LIN {X -94.212,Y -11.587,Z -73.659,A -90.000,B 90.000,C 0.000} C_DIS
LIN {X -94.293,Y -11.592,Z -73.648,A -90.000,B 90.000,C 0.000} C_DIS
LIN {X -94.845,Y -11.615,Z -73.582,A -90.000,B 90.000,C 0.000} C_DIS
LIN {X -95.072,Y -11.619,Z -73.546,A -90.000,B 90.000,C 0.000} C_DIS
LIN {X -95.448,Y -11.620,Z -73.492,A -90.000,B 90.000,C 0.000} C_DIS
LIN {X -95.686,Y -11.622,Z -73.458,A -90.000,B 90.000,C 0.000} C_DIS
LIN {X -96.285,Y -11.645,Z -73.361,A -90.000,B 90.000,C 0.000} C_DIS
LIN {X -96.529,Y -11.657,Z -73.323,A -90.000,B 90.000,C 0.000} C_DIS
LIN {X -96.718,Y -11.655,Z -73.288,A -90.000,B 90.000,C 0.000} C_DIS
LIN {X -97.124,Y -11.644,Z -73.202,A -90.000,B 90.000,C 0.000} C_DIS
LIN {X -97.511,Y -11.644,Z -73.113,A -90.000,B 90.000,C 0.000} C_DIS
LIN {X -97.707,Y -11.652,Z -73.075,A -90.000,B 90.000,C 0.000} C_DIS
LIN {X -98.138,Y -11.663,Z -72.965,A -90.000,B 90.000,C 0.000} C_DIS
LIN {X -98.421,Y -11.660,Z -72.876,A -90.000,B 90.000,C 0.000} C_DIS
LIN {X -98.629,Y -11.654,Z -72.804,A -90.000,B 90.000,C 0.000} C_DIS
LIN {X -98.764,Y -11.646,Z -72.759,A -90.000,B 90.000,C 0.000} C_DIS
LIN {X -98.907,Y -11.642,Z -72.709,A -90.000,B 90.000,C 0.000} C_DIS
LIN {X -99.025,Y -11.642,Z -72.667,A -90.000,B 90.000,C 0.000} C_DIS
LIN {X -99.303,Y -11.649,Z -72.577,A -90.000,B 90.000,C 0.000} C_DIS
LIN {X -99.385,Y -11.652,Z -72.549,A -90.000,B 90.000,C 0.000} C_DIS
LIN {X -99.802,Y -11.664,Z -72.390,A -90.000,B 90.000,C 0.000} C_DIS
LIN {X -100.084,Y -11.662,Z -72.264,A -90.000,B 90.000,C 0.000} C_DIS
LIN {X -100.297,Y -11.652,Z -72.158,A -90.000,B 90.000,C 0.000} C_DIS
LIN {X -100.506,Y -11.637,Z -72.058,A -90.000,B 90.000,C 0.000} C_DIS
LIN {X -100.618,Y -11.632,Z -72.002,A -90.000,B 90.000,C 0.000} C_DIS
LIN {X -101.008,Y -11.626,Z -71.798,A -90.000,B 90.000,C 0.000} C_DIS
LIN {X -101.217,Y -11.633,Z -71.690,A -90.000,B 90.000,C 0.000} C_DIS
LIN {X -101.505,Y -11.645,Z -71.539,A -90.000,B 90.000,C 0.000} C_DIS
LIN {X -101.784,Y -11.648,Z -71.377,A -90.000,B 90.000,C 0.000} C_DIS
LIN {X -102.159,Y -11.635,Z -71.132,A -90.000,B 90.000,C 0.000} C_DIS
LIN {X -102.376,Y -11.622,Z -70.990,A -90.000,B 90.000,C 0.000} C_DIS
LIN {X -102.782,Y -11.607,Z -70.696,A -90.000,B 90.000,C 0.000} C_DIS
LIN {X -102.971,Y -11.606,Z -70.555,A -90.000,B 90.000,C 0.000} C_DIS
LIN {X -103.503,Y -11.618,Z -70.146,A -90.000,B 90.000,C 0.000} C_DIS
LIN {X -103.891,Y -11.613,Z -69.818,A -90.000,B 90.000,C 0.000} C_DIS
LIN {X -104.471,Y -11.591,Z -69.295,A -90.000,B 90.000,C 0.000} C_DIS
LIN {X -104.553,Y -11.591,Z -69.219,A -90.000,B 90.000,C 0.000} C_DIS
LIN {X -104.963,Y -11.602,Z -68.827,A -90.000,B 90.000,C 0.000} C_DIS
LIN {X -105.136,Y -11.603,Z -68.655,A -90.000,B 90.000,C 0.000} C_DIS
LIN {X -105.249,Y -11.602,Z -68.539,A -90.000,B 90.000,C 0.000} C_DIS
LIN {X -105.573,Y -11.597,Z -68.197,A -90.000,B 90.000,C 0.000} C_DIS
LIN {X -105.950,Y -11.592,Z -67.792,A -90.000,B 90.000,C 0.000} C_DIS
LIN {X -106.246,Y -11.591,Z -67.471,A -90.000,B 90.000,C 0.000} C_DIS
LIN {X -106.503,Y -11.591,Z -67.178,A -90.000,B 90.000,C 0.000} C_DIS
LIN {X -106.747,Y -11.594,Z -66.899,A -90.000,B 90.000,C 0.000} C_DIS
LIN {X -107.149,Y -11.591,Z -66.405,A -90.000,B 90.000,C 0.000} C_DIS
LIN {X -107.576,Y -11.586,Z -65.870,A -90.000,B 90.000,C 0.000} C_DIS
LIN {X -107.870,Y -11.590,Z -65.494,A -90.000,B 90.000,C 0.000} C_DIS
LIN {X -108.183,Y -11.592,Z -65.074,A -90.000,B 90.000,C 0.000} C_DIS
LIN {X -108.727,Y -11.597,Z -64.294,A -90.000,B 90.000,C 0.000} C_DIS
LIN {X -108.884,Y -11.600,Z -64.066,A -90.000,B 90.000,C 0.000} C_DIS
LIN {X -109.086,Y -11.609,Z -63.770,A -90.000,B 90.000,C 0.000} C_DIS
LIN {X -109.795,Y -11.609,Z -62.636,A -90.000,B 90.000,C 0.000} C_DIS
LIN {X -109.878,Y -11.610,Z -62.503,A -90.000,B 90.000,C 0.000} C_DIS
LIN {X -109.980,Y -11.610,Z -62.332,A -90.000,B 90.000,C 0.000} C_DIS
LIN {X -110.151,Y -11.614,Z -62.039,A -90.000,B 90.000,C 0.000} C_DIS
LIN {X -110.277,Y -11.619,Z -61.794,A -90.000,B 90.000,C 0.000} C_DIS
LIN {X -110.690,Y -11.621,Z -60.933,A -90.000,B 90.000,C 0.000} C_DIS
LIN {X -110.735,Y -11.626,Z -60.833,A -90.000,B 90.000,C 0.000} C_DIS
LIN {X -110.921,Y -11.645,Z -60.397,A -90.000,B 90.000,C 0.000} C_DIS
LIN {X -111.213,Y -11.660,Z -59.639,A -90.000,B 90.000,C 0.000} C_DIS
LIN {X -111.406,Y -11.675,Z -59.133,A -90.000,B 90.000,C 0.000} C_DIS
LIN {X -111.465,Y -11.679,Z -58.954,A -90.000,B 90.000,C 0.000} C_DIS
LIN {X -111.561,Y -11.684,Z -58.654,A -90.000,B 90.000,C 0.000} C_DIS
LIN {X -111.600,Y -11.686,Z -58.518,A -90.000,B 90.000,C 0.000} C_DIS
LIN {X -111.705,Y -11.680,Z -58.092,A -90.000,B 90.000,C 0.000} C_DIS
LIN {X -111.798,Y -11.682,Z -57.690,A -90.000,B 90.000,C 0.000} C_DIS
LIN {X -111.872,Y -11.683,Z -57.324,A -90.000,B 90.000,C 0.000} C_DIS
LIN {X -111.987,Y -11.695,Z -56.667,A -90.000,B 90.000,C 0.000} C_DIS
LIN {X -112.103,Y -11.699,Z -56.102,A -90.000,B 90.000,C 0.000} C_DIS
LIN {X -112.133,Y -11.705,Z -55.941,A -90.000,B 90.000,C 0.000} C_DIS
LIN {X -112.214,Y -11.706,Z -55.543,A -90.000,B 90.000,C 0.000} C_DIS
LIN {X -112.258,Y -11.710,Z -55.310,A -90.000,B 90.000,C 0.000} C_DIS
LIN {X -112.301,Y -11.709,Z -55.111,A -90.000,B 90.000,C 0.000} C_DIS
LIN {X -112.331,Y -11.710,Z -54.963,A -90.000,B 90.000,C 0.000} C_DIS
LIN {X -112.384,Y -11.700,Z -54.736,A -90.000,B 90.000,C 0.000} C_DIS
LIN {X -112.413,Y -11.683,Z -54.654,A -90.000,B 90.000,C 0.000} C_DIS
LIN {X -112.468,Y -11.659,Z -54.515,A -90.000,B 90.000,C 0.000} C_DIS
LIN {X -112.573,Y -11.623,Z -54.266,A -90.000,B 90.000,C 0.000} C_DIS
LIN {X -112.724,Y -11.568,Z -53.872,A -90.000,B 90.000,C 0.000} C_DIS
LIN {X -112.828,Y -11.542,Z -53.616,A -90.000,B 90.000,C 0.000} C_DIS
LIN {X -112.987,Y -11.505,Z -53.211,A -90.000,B 90.000,C 0.000} C_DIS
LIN {X -113.167,Y -11.475,Z -52.722,A -90.000,B 90.000,C 0.000} C_DIS
LIN {X -113.273,Y -11.462,Z -52.423,A -90.000,B 90.000,C 0.000} C_DIS
LIN {X -113.396,Y -11.439,Z -52.007,A -90.000,B 90.000,C 0.000} C_DIS
LIN {X -113.436,Y -11.433,Z -51.874,A -90.000,B 90.000,C 0.000} C_DIS
LIN {X -113.514,Y -11.415,Z -51.552,A -90.000,B 90.000,C 0.000} C_DIS
LIN {X -113.736,Y -11.433,Z -51.065,A -90.000,B 90.000,C 0.000} C_DIS
LIN {X -113.844,Y -11.447,Z -50.817,A -90.000,B 90.000,C 0.000} C_DIS
LIN {X -113.954,Y -11.459,Z -50.527,A -90.000,B 90.000,C 0.000} C_DIS
LIN {X -114.109,Y -11.480,Z -50.102,A -90.000,B 90.000,C 0.000} C_DIS
LIN {X -114.142,Y -11.486,Z -50.008,A -90.000,B 90.000,C 0.000} C_DIS
LIN {X -114.248,Y -11.503,Z -49.683,A -90.000,B 90.000,C 0.000} C_DIS
LIN {X -114.317,Y -11.524,Z -49.458,A -90.000,B 90.000,C 0.000} C_DIS
LIN {X -114.400,Y -11.549,Z -49.090,A -90.000,B 90.000,C 0.000} C_DIS
LIN {X -114.487,Y -11.577,Z -48.657,A -90.000,B 90.000,C 0.000} C_DIS
LIN {X -114.535,Y -11.593,Z -48.376,A -90.000,B 90.000,C 0.000} C_DIS
LIN {X -114.551,Y -11.601,Z -48.274,A -90.000,B 90.000,C 0.000} C_DIS
LIN {X -114.562,Y -11.609,Z -48.204,A -90.000,B 90.000,C 0.000} C_DIS
LIN {X -114.587,Y -11.631,Z -47.823,A -90.000,B 90.000,C 0.000} C_DIS
LIN {X -114.597,Y -11.652,Z -47.585,A -90.000,B 90.000,C 0.000} C_DIS
LIN {X -114.602,Y -11.671,Z -47.417,A -90.000,B 90.000,C 0.000} C_DIS
LIN {X -114.599,Y -11.700,Z -47.076,A -90.000,B 90.000,C 0.000} C_DIS
LIN {X -114.573,Y -11.723,Z -46.648,A -90.000,B 90.000,C 0.000} C_DIS
LIN {X -114.555,Y -11.731,Z -46.497,A -90.000,B 90.000,C 0.000} C_DIS
LIN {X -114.524,Y -11.750,Z -46.285,A -90.000,B 90.000,C 0.000} C_DIS
LIN {X -114.446,Y -11.774,Z -45.861,A -90.000,B 90.000,C 0.000} C_DIS
LIN {X -114.403,Y -11.785,Z -45.648,A -90.000,B 90.000,C 0.000} C_DIS
LIN {X -114.366,Y -11.793,Z -45.512,A -90.000,B 90.000,C 0.000} C_DIS
LIN {X -114.304,Y -11.811,Z -45.294,A -90.000,B 90.000,C 0.000} C_DIS
LIN {X -114.182,Y -11.836,Z -44.903,A -90.000,B 90.000,C 0.000} C_DIS
LIN {X -114.168,Y -11.836,Z -44.865,A -90.000,B 90.000,C 0.000} C_DIS
LIN {X -114.169,Y -11.819,Z -44.821,A -90.000,B 90.000,C 0.000} C_DIS
LIN {X -114.168,Y -11.721,Z -44.547,A -90.000,B 90.000,C 0.000} C_DIS
LIN {X -114.165,Y -11.685,Z -44.438,A -90.000,B 90.000,C 0.000} C_DIS
LIN {X -114.151,Y -11.619,Z -44.239,A -90.000,B 90.000,C 0.000} C_DIS
LIN {X -114.122,Y -11.537,Z -43.961,A -90.000,B 90.000,C 0.000} C_DIS
LIN {X -114.106,Y -11.508,Z -43.858,A -90.000,B 90.000,C 0.000} C_DIS
LIN {X -114.085,Y -11.479,Z -43.749,A -90.000,B 90.000,C 0.000} C_DIS
LIN {X -114.038,Y -11.429,Z -43.536,A -90.000,B 90.000,C 0.000} C_DIS
LIN {X -114.035,Y -11.426,Z -43.521,A -90.000,B 90.000,C 0.000} C_DIS
LIN {X -114.241,Y -11.433,Z -43.054,A -90.000,B 90.000,C 0.000} C_DIS
LIN {X -114.306,Y -11.437,Z -42.901,A -90.000,B 90.000,C 0.000} C_DIS
LIN {X -114.518,Y -11.448,Z -42.384,A -90.000,B 90.000,C 0.000} C_DIS
LIN {X -114.643,Y -11.454,Z -42.061,A -90.000,B 90.000,C 0.000} C_DIS
LIN {X -114.710,Y -11.459,Z -41.886,A -90.000,B 90.000,C 0.000} C_DIS
LIN {X -114.857,Y -11.470,Z -41.484,A -90.000,B 90.000,C 0.000} C_DIS
LIN {X -115.017,Y -11.486,Z -40.978,A -90.000,B 90.000,C 0.000} C_DIS
LIN {X -115.171,Y -11.505,Z -40.471,A -90.000,B 90.000,C 0.000} C_DIS
LIN {X -115.237,Y -11.511,Z -40.206,A -90.000,B 90.000,C 0.000} C_DIS
LIN {X -115.269,Y -11.516,Z -40.071,A -90.000,B 90.000,C 0.000} C_DIS
LIN {X -115.346,Y -11.529,Z -39.718,A -90.000,B 90.000,C 0.000} C_DIS
LIN {X -115.399,Y -11.542,Z -39.436,A -90.000,B 90.000,C 0.000} C_DIS
LIN {X -115.423,Y -11.547,Z -39.289,A -90.000,B 90.000,C 0.000} C_DIS
LIN {X -115.469,Y -11.553,Z -38.903,A -90.000,B 90.000,C 0.000} C_DIS
LIN {X -115.487,Y -11.558,Z -38.743,A -90.000,B 90.000,C 0.000} C_DIS
LIN {X -115.510,Y -11.568,Z -38.507,A -90.000,B 90.000,C 0.000} C_DIS
LIN {X -115.536,Y -11.587,Z -38.116,A -90.000,B 90.000,C 0.000} C_DIS
LIN {X -115.547,Y -11.598,Z -37.805,A -90.000,B 90.000,C 0.000} C_DIS
LIN {X -115.546,Y -11.599,Z -37.768,A -90.000,B 90.000,C 0.000} C_DIS
LIN {X -115.535,Y -11.611,Z -37.401,A -90.000,B 90.000,C 0.000} C_DIS
LIN {X -115.517,Y -11.629,Z -37.064,A -90.000,B 90.000,C 0.000} C_DIS
LIN {X -115.474,Y -11.636,Z -36.708,A -90.000,B 90.000,C 0.000} C_DIS
LIN {X -115.454,Y -11.640,Z -36.570,A -90.000,B 90.000,C 0.000} C_DIS
LIN {X -115.407,Y -11.656,Z -36.278,A -90.000,B 90.000,C 0.000} C_DIS
LIN {X -115.349,Y -11.665,Z -35.994,A -90.000,B 90.000,C 0.000} C_DIS
LIN {X -115.297,Y -11.669,Z -35.782,A -90.000,B 90.000,C 0.000} C_DIS
LIN {X -115.179,Y -11.680,Z -35.351,A -90.000,B 90.000,C 0.000} C_DIS
LIN {X -115.107,Y -11.690,Z -35.107,A -90.000,B 90.000,C 0.000} C_DIS
LIN {X -115.003,Y -11.696,Z -34.808,A -90.000,B 90.000,C 0.000} C_DIS
LIN {X -114.904,Y -11.698,Z -34.550,A -90.000,B 90.000,C 0.000} C_DIS
LIN {X -114.796,Y -11.706,Z -34.283,A -90.000,B 90.000,C 0.000} C_DIS
LIN {X -114.748,Y -11.712,Z -34.170,A -90.000,B 90.000,C 0.000} C_DIS
LIN {X -114.623,Y -11.720,Z -33.910,A -90.000,B 90.000,C 0.000} C_DIS
LIN {X -114.429,Y -11.726,Z -33.544,A -90.000,B 90.000,C 0.000} C_DIS
LIN {X -114.375,Y -11.729,Z -33.450,A -90.000,B 90.000,C 0.000} C_DIS
LIN {X -114.266,Y -11.737,Z -33.272,A -90.000,B 90.000,C 0.000} C_DIS
LIN {X -114.093,Y -11.740,Z -33.018,A -90.000,B 90.000,C 0.000} C_DIS
LIN {X -114.019,Y -11.742,Z -32.909,A -90.000,B 90.000,C 0.000} C_DIS
LIN {X -113.928,Y -11.743,Z -32.783,A -90.000,B 90.000,C 0.000} C_DIS
LIN {X -113.839,Y -11.749,Z -32.668,A -90.000,B 90.000,C 0.000} C_DIS
LIN {X -113.552,Y -11.754,Z -32.335,A -90.000,B 90.000,C 0.000} C_DIS
LIN {X -113.377,Y -11.754,Z -32.146,A -90.000,B 90.000,C 0.000} C_DIS
LIN {X -113.255,Y -11.757,Z -32.021,A -90.000,B 90.000,C 0.000} C_DIS
LIN {X -112.860,Y -11.759,Z -31.635,A -90.000,B 90.000,C 0.000} C_DIS
LIN {X -112.787,Y -11.754,Z -31.554,A -90.000,B 90.000,C 0.000} C_DIS
LIN {X -112.743,Y -11.754,Z -31.498,A -90.000,B 90.000,C 0.000} C_DIS
LIN {X -112.607,Y -11.754,Z -31.317,A -90.000,B 90.000,C 0.000} C_DIS
LIN {X -112.172,Y -11.764,Z -30.704,A -90.000,B 90.000,C 0.000} C_DIS
LIN {X -112.046,Y -11.772,Z -30.531,A -90.000,B 90.000,C 0.000} C_DIS
LIN {X -111.786,Y -11.780,Z -30.189,A -90.000,B 90.000,C 0.000} C_DIS
LIN {X -111.636,Y -11.792,Z -29.999,A -90.000,B 90.000,C 0.000} C_DIS
LIN {X -111.260,Y -11.802,Z -29.560,A -90.000,B 90.000,C 0.000} C_DIS
LIN {X -111.118,Y -11.804,Z -29.402,A -90.000,B 90.000,C 0.000} C_DIS
LIN {X -111.007,Y -11.810,Z -29.282,A -90.000,B 90.000,C 0.000} C_DIS
LIN {X -110.702,Y -11.818,Z -28.964,A -90.000,B 90.000,C 0.000} C_DIS
LIN {X -110.630,Y -11.822,Z -28.890,A -90.000,B 90.000,C 0.000} C_DIS
LIN {X -110.226,Y -11.831,Z -28.505,A -90.000,B 90.000,C 0.000} C_DIS
LIN {X -109.683,Y -11.835,Z -28.022,A -90.000,B 90.000,C 0.000} C_DIS
LIN {X -109.483,Y -11.838,Z -27.846,A -90.000,B 90.000,C 0.000} C_DIS
LIN {X -109.036,Y -11.838,Z -27.473,A -90.000,B 90.000,C 0.000} C_DIS
LIN {X -108.440,Y -11.835,Z -27.051,A -90.000,B 90.000,C 0.000} C_DIS
LIN {X -108.173,Y -11.837,Z -26.866,A -90.000,B 90.000,C 0.000} C_DIS
LIN {X -108.077,Y -11.832,Z -26.807,A -90.000,B 90.000,C 0.000} C_DIS
LIN {X -107.401,Y -11.827,Z -26.429,A -90.000,B 90.000,C 0.000} C_DIS
LIN {X -107.170,Y -11.828,Z -26.305,A -90.000,B 90.000,C 0.000} C_DIS
LIN {X -106.974,Y -11.818,Z -26.212,A -90.000,B 90.000,C 0.000} C_DIS
LIN {X -106.880,Y -11.816,Z -26.170,A -90.000,B 90.000,C 0.000} C_DIS
LIN {X -106.375,Y -11.813,Z -25.952,A -90.000,B 90.000,C 0.000} C_DIS
LIN {X -106.083,Y -11.808,Z -25.832,A -90.000,B 90.000,C 0.000} C_DIS
LIN {X -105.983,Y -11.808,Z -25.792,A -90.000,B 90.000,C 0.000} C_DIS
LIN {X -105.685,Y -11.798,Z -25.686,A -90.000,B 90.000,C 0.000} C_DIS
LIN {X -105.383,Y -11.796,Z -25.586,A -90.000,B 90.000,C 0.000} C_DIS
LIN {X -104.972,Y -11.796,Z -25.452,A -90.000,B 90.000,C 0.000} C_DIS
LIN {X -104.611,Y -11.788,Z -25.344,A -90.000,B 90.000,C 0.000} C_DIS
LIN {X -103.526,Y -11.781,Z -25.036,A -90.000,B 90.000,C 0.000} C_DIS
LIN {X -103.108,Y -11.775,Z -24.918,A -90.000,B 90.000,C 0.000} C_DIS
LIN {X -102.960,Y -11.719,Z -24.832,A -90.000,B 90.000,C 0.000} C_DIS
LIN {X -102.802,Y -11.666,Z -24.747,A -90.000,B 90.000,C 0.000} C_DIS
LIN {X -102.662,Y -11.616,Z -24.668,A -90.000,B 90.000,C 0.000} C_DIS
LIN {X -102.539,Y -11.576,Z -24.600,A -90.000,B 90.000,C 0.000} C_DIS
LIN {X -102.363,Y -11.527,Z -24.507,A -90.000,B 90.000,C 0.000} C_DIS
LIN {X -102.114,Y -11.465,Z -24.383,A -90.000,B 90.000,C 0.000} C_DIS
LIN {X -102.014,Y -11.483,Z -24.180,A -90.000,B 90.000,C 0.000} C_DIS
LIN {X -101.901,Y -11.496,Z -23.951,A -90.000,B 90.000,C 0.000} C_DIS
LIN {X -101.819,Y -11.510,Z -23.792,A -90.000,B 90.000,C 0.000} C_DIS
LIN {X -101.710,Y -11.525,Z -23.594,A -90.000,B 90.000,C 0.000} C_DIS
LIN {X -101.650,Y -11.538,Z -23.477,A -90.000,B 90.000,C 0.000} C_DIS
LIN {X -101.419,Y -11.566,Z -23.099,A -90.000,B 90.000,C 0.000} C_DIS
LIN {X -101.286,Y -11.578,Z -22.907,A -90.000,B 90.000,C 0.000} C_DIS
LIN {X -101.230,Y -11.582,Z -22.829,A -90.000,B 90.000,C 0.000} C_DIS
LIN {X -101.083,Y -11.591,Z -22.633,A -90.000,B 90.000,C 0.000} C_DIS
LIN {X -100.905,Y -11.613,Z -22.406,A -90.000,B 90.000,C 0.000} C_DIS
LIN {X -100.650,Y -11.640,Z -22.107,A -90.000,B 90.000,C 0.000} C_DIS
LIN {X -100.625,Y -11.641,Z -22.081,A -90.000,B 90.000,C 0.000} C_DIS
LIN {X -100.490,Y -11.647,Z -21.949,A -90.000,B 90.000,C 0.000} C_DIS
LIN {X -100.295,Y -11.662,Z -21.766,A -90.000,B 90.000,C 0.000} C_DIS
LIN {X -100.058,Y -11.673,Z -21.577,A -90.000,B 90.000,C 0.000} C_DIS
LIN {X -99.895,Y -11.680,Z -21.451,A -90.000,B 90.000,C 0.000} C_DIS
LIN {X -99.709,Y -11.695,Z -21.311,A -90.000,B 90.000,C 0.000} C_DIS
LIN {X -99.552,Y -11.703,Z -21.207,A -90.000,B 90.000,C 0.000} C_DIS
LIN {X -99.332,Y -11.712,Z -21.073,A -90.000,B 90.000,C 0.000} C_DIS
LIN {X -99.161,Y -11.716,Z -20.976,A -90.000,B 90.000,C 0.000} C_DIS
LIN {X -99.058,Y -11.719,Z -20.926,A -90.000,B 90.000,C 0.000} C_DIS
LIN {X -98.927,Y -11.725,Z -20.865,A -90.000,B 90.000,C 0.000} C_DIS
LIN {X -98.675,Y -11.730,Z -20.758,A -90.000,B 90.000,C 0.000} C_DIS
LIN {X -98.528,Y -11.739,Z -20.699,A -90.000,B 90.000,C 0.000} C_DIS
LIN {X -98.215,Y -11.762,Z -20.586,A -90.000,B 90.000,C 0.000} C_DIS
LIN {X -97.800,Y -11.772,Z -20.465,A -90.000,B 90.000,C 0.000} C_DIS
LIN {X -97.726,Y -11.774,Z -20.449,A -90.000,B 90.000,C 0.000} C_DIS
LIN {X -97.685,Y -11.782,Z -20.434,A -90.000,B 90.000,C 0.000} C_DIS
LIN {X -97.660,Y -11.787,Z -20.423,A -90.000,B 90.000,C 0.000} C_DIS
LIN {X -97.342,Y -11.881,Z -20.275,A -90.000,B 90.000,C 0.000} C_DIS
LIN {X -97.307,Y -11.894,Z -20.257,A -90.000,B 90.000,C 0.000} C_DIS
LIN {X -97.142,Y -11.960,Z -20.180,A -90.000,B 90.000,C 0.000} C_DIS
LIN {X -97.021,Y -12.013,Z -20.130,A -90.000,B 90.000,C 0.000} C_DIS
LIN {X -96.913,Y -11.978,Z -19.972,A -90.000,B 90.000,C 0.000} C_DIS
LIN {X -96.868,Y -11.963,Z -19.913,A -90.000,B 90.000,C 0.000} C_DIS
LIN {X -96.756,Y -11.939,Z -19.760,A -90.000,B 90.000,C 0.000} C_DIS
LIN {X -96.712,Y -11.932,Z -19.703,A -90.000,B 90.000,C 0.000} C_DIS
LIN {X -96.487,Y -11.886,Z -19.438,A -90.000,B 90.000,C 0.000} C_DIS
LIN {X -96.353,Y -11.867,Z -19.275,A -90.000,B 90.000,C 0.000} C_DIS
LIN {X -96.154,Y -11.834,Z -19.045,A -90.000,B 90.000,C 0.000} C_DIS
LIN {X -96.089,Y -11.826,Z -18.977,A -90.000,B 90.000,C 0.000} C_DIS
LIN {X -95.848,Y -11.806,Z -18.731,A -90.000,B 90.000,C 0.000} C_DIS
LIN {X -95.599,Y -11.777,Z -18.499,A -90.000,B 90.000,C 0.000} C_DIS
LIN {X -95.498,Y -11.769,Z -18.409,A -90.000,B 90.000,C 0.000} C_DIS
LIN {X -95.397,Y -11.763,Z -18.324,A -90.000,B 90.000,C 0.000} C_DIS
LIN {X -95.266,Y -11.753,Z -18.219,A -90.000,B 90.000,C 0.000} C_DIS
LIN {X -95.101,Y -11.743,Z -18.088,A -90.000,B 90.000,C 0.000} C_DIS
LIN {X -94.938,Y -11.726,Z -17.971,A -90.000,B 90.000,C 0.000} C_DIS
LIN {X -94.819,Y -11.719,Z -17.890,A -90.000,B 90.000,C 0.000} C_DIS
LIN {X -94.307,Y -11.706,Z -17.553,A -90.000,B 90.000,C 0.000} C_DIS
LIN {X -93.957,Y -11.677,Z -17.360,A -90.000,B 90.000,C 0.000} C_DIS
LIN {X -93.803,Y -11.670,Z -17.281,A -90.000,B 90.000,C 0.000} C_DIS
LIN {X -93.404,Y -11.650,Z -17.099,A -90.000,B 90.000,C 0.000} C_DIS
LIN {X -93.140,Y -11.647,Z -16.984,A -90.000,B 90.000,C 0.000} C_DIS
LIN {X -92.940,Y -11.639,Z -16.907,A -90.000,B 90.000,C 0.000} C_DIS
LIN {X -92.233,Y -11.605,Z -16.673,A -90.000,B 90.000,C 0.000} C_DIS
LIN {X -92.077,Y -11.601,Z -16.623,A -90.000,B 90.000,C 0.000} C_DIS
LIN {X -91.780,Y -11.599,Z -16.539,A -90.000,B 90.000,C 0.000} C_DIS
LIN {X -91.315,Y -11.579,Z -16.439,A -90.000,B 90.000,C 0.000} C_DIS
LIN {X -90.900,Y -11.559,Z -16.359,A -90.000,B 90.000,C 0.000} C_DIS
LIN {X -90.731,Y -11.553,Z -16.329,A -90.000,B 90.000,C 0.000} C_DIS
LIN {X -90.367,Y -11.549,Z -16.267,A -90.000,B 90.000,C 0.000} C_DIS
LIN {X -90.191,Y -11.544,Z -16.249,A -90.000,B 90.000,C 0.000} C_DIS
LIN {X -89.833,Y -11.536,Z -16.216,A -90.000,B 90.000,C 0.000} C_DIS
LIN {X -89.165,Y -11.518,Z -16.171,A -90.000,B 90.000,C 0.000} C_DIS
LIN {X -88.792,Y -11.516,Z -16.148,A -90.000,B 90.000,C 0.000} C_DIS
LIN {X -88.664,Y -11.513,Z -16.145,A -90.000,B 90.000,C 0.000} C_DIS
LIN {X -87.183,Y -11.506,Z -16.212,A -90.000,B 90.000,C 0.000} C_DIS
LIN {X -87.099,Y -11.505,Z -16.218,A -90.000,B 90.000,C 0.000} C_DIS
LIN {X -86.917,Y -11.502,Z -16.245,A -90.000,B 90.000,C 0.000} C_DIS
LIN {X -86.828,Y -11.544,Z -16.175,A -90.000,B 90.000,C 0.000} C_DIS
LIN {X -86.636,Y -11.536,Z -15.957,A -90.000,B 90.000,C 0.000} C_DIS
LIN {X -86.604,Y -11.535,Z -15.920,A -90.000,B 90.000,C 0.000} C_DIS
LIN {X -86.521,Y -11.528,Z -15.838,A -90.000,B 90.000,C 0.000} C_DIS
LIN {X -86.433,Y -11.522,Z -15.756,A -90.000,B 90.000,C 0.000} C_DIS
LIN {X -86.245,Y -11.516,Z -15.585,A -90.000,B 90.000,C 0.000} C_DIS
LIN {X -86.143,Y -11.511,Z -15.498,A -90.000,B 90.000,C 0.000} C_DIS
LIN {X -86.001,Y -11.505,Z -15.384,A -90.000,B 90.000,C 0.000} C_DIS
LIN {X -85.716,Y -11.501,Z -15.165,A -90.000,B 90.000,C 0.000} C_DIS
LIN {X -85.489,Y -11.497,Z -15.001,A -90.000,B 90.000,C 0.000} C_DIS
LIN {X -85.292,Y -11.490,Z -14.870,A -90.000,B 90.000,C 0.000} C_DIS
LIN {X -85.056,Y -11.485,Z -14.730,A -90.000,B 90.000,C 0.000} C_DIS
LIN {X -84.838,Y -11.476,Z -14.614,A -90.000,B 90.000,C 0.000} C_DIS
LIN {X -84.643,Y -11.474,Z -14.512,A -90.000,B 90.000,C 0.000} C_DIS
LIN {X -84.496,Y -11.471,Z -14.444,A -90.000,B 90.000,C 0.000} C_DIS
LIN {X -84.276,Y -11.471,Z -14.336,A -90.000,B 90.000,C 0.000} C_DIS
LIN {X -83.945,Y -11.460,Z -14.203,A -90.000,B 90.000,C 0.000} C_DIS
LIN {X -83.789,Y -11.458,Z -14.143,A -90.000,B 90.000,C 0.000} C_DIS
LIN {X -83.679,Y -11.457,Z -14.101,A -90.000,B 90.000,C 0.000} C_DIS
LIN {X -83.236,Y -11.440,Z -13.976,A -90.000,B 90.000,C 0.000} C_DIS
LIN {X -82.907,Y -11.438,Z -13.879,A -90.000,B 90.000,C 0.000} C_DIS
LIN {X -82.511,Y -11.435,Z -13.771,A -90.000,B 90.000,C 0.000} C_DIS
LIN {X -82.198,Y -11.423,Z -13.716,A -90.000,B 90.000,C 0.000} C_DIS
LIN {X -81.975,Y -11.420,Z -13.678,A -90.000,B 90.000,C 0.000} C_DIS
LIN {X -81.855,Y -11.418,Z -13.660,A -90.000,B 90.000,C 0.000} C_DIS
LIN {X -81.523,Y -11.419,Z -13.594,A -90.000,B 90.000,C 0.000} C_DIS
LIN {X -81.089,Y -11.414,Z -13.523,A -90.000,B 90.000,C 0.000} C_DIS
LIN {X -81.051,Y -11.414,Z -13.517,A -90.000,B 90.000,C 0.000} C_DIS
LIN {X -80.708,Y -11.410,Z -13.483,A -90.000,B 90.000,C 0.000} C_DIS
LIN {X -80.352,Y -11.408,Z -13.451,A -90.000,B 90.000,C 0.000} C_DIS
LIN {X -80.279,Y -11.409,Z -13.442,A -90.000,B 90.000,C 0.000} C_DIS
LIN {X -79.938,Y -11.409,Z -13.401,A -90.000,B 90.000,C 0.000} C_DIS
LIN {X -79.461,Y -11.404,Z -13.374,A -90.000,B 90.000,C 0.000} C_DIS
LIN {X -78.870,Y -11.401,Z -13.362,A -90.000,B 90.000,C 0.000} C_DIS
LIN {X -78.618,Y -11.401,Z -13.361,A -90.000,B 90.000,C 0.000} C_DIS
LIN {X -78.465,Y -11.401,Z -13.358,A -90.000,B 90.000,C 0.000} C_DIS
LIN {X -78.196,Y -11.400,Z -13.367,A -90.000,B 90.000,C 0.000} C_DIS
LIN {X -77.753,Y -11.395,Z -13.389,A -90.000,B 90.000,C 0.000} C_DIS
LIN {X -77.193,Y -11.394,Z -13.435,A -90.000,B 90.000,C 0.000} C_DIS
LIN {X -76.796,Y -11.393,Z -13.491,A -90.000,B 90.000,C 0.000} C_DIS
LIN {X -76.319,Y -11.389,Z -13.573,A -90.000,B 90.000,C 0.000} C_DIS
LIN {X -75.821,Y -11.382,Z -13.682,A -90.000,B 90.000,C 0.000} C_DIS
LIN {X -75.289,Y -11.380,Z -13.800,A -90.000,B 90.000,C 0.000} C_DIS
LIN {X -74.826,Y -11.378,Z -13.931,A -90.000,B 90.000,C 0.000} C_DIS
LIN {X -74.667,Y -11.378,Z -13.978,A -90.000,B 90.000,C 0.000} C_DIS
LIN {X -74.204,Y -11.368,Z -14.158,A -90.000,B 90.000,C 0.000} C_DIS
LIN {X -73.840,Y -11.362,Z -14.305,A -90.000,B 90.000,C 0.000} C_DIS
LIN {X -73.396,Y -11.359,Z -14.469,A -90.000,B 90.000,C 0.000} C_DIS
LIN {X -72.945,Y -11.354,Z -14.648,A -90.000,B 90.000,C 0.000} C_DIS
LIN {X -72.686,Y -11.351,Z -14.763,A -90.000,B 90.000,C 0.000} C_DIS
LIN {X -72.170,Y -11.349,Z -14.974,A -90.000,B 90.000,C 0.000} C_DIS
LIN {X -71.784,Y -11.353,Z -15.134,A -90.000,B 90.000,C 0.000} C_DIS
LIN {X -71.617,Y -11.355,Z -15.206,A -90.000,B 90.000,C 0.000} C_DIS
LIN {X -70.795,Y -11.358,Z -15.576,A -90.000,B 90.000,C 0.000} C_DIS
LIN {X -69.979,Y -11.366,Z -15.948,A -90.000,B 90.000,C 0.000} C_DIS
LIN {X -69.569,Y -11.371,Z -16.140,A -90.000,B 90.000,C 0.000} C_DIS
LIN {X -68.609,Y -11.381,Z -16.596,A -90.000,B 90.000,C 0.000} C_DIS
LIN {X -68.413,Y -11.382,Z -16.694,A -90.000,B 90.000,C 0.000} C_DIS
LIN {X -67.117,Y -11.397,Z -17.317,A -90.000,B 90.000,C 0.000} C_DIS
LIN {X -66.418,Y -11.408,Z -17.647,A -90.000,B 90.000,C 0.000} C_DIS
LIN {X -65.864,Y -11.416,Z -17.911,A -90.000,B 90.000,C 0.000} C_DIS
LIN {X -65.636,Y -11.422,Z -18.020,A -90.000,B 90.000,C 0.000} C_DIS
LIN {X -65.398,Y -11.430,Z -18.128,A -90.000,B 90.000,C 0.000} C_DIS
LIN {X -64.927,Y -11.436,Z -18.340,A -90.000,B 90.000,C 0.000} C_DIS
LIN {X -64.688,Y -11.444,Z -18.450,A -90.000,B 90.000,C 0.000} C_DIS
LIN {X -64.411,Y -11.451,Z -18.586,A -90.000,B 90.000,C 0.000} C_DIS
LIN {X -64.115,Y -11.463,Z -18.716,A -90.000,B 90.000,C 0.000} C_DIS
LIN {X -63.630,Y -11.473,Z -18.925,A -90.000,B 90.000,C 0.000} C_DIS
LIN {X -63.453,Y -11.477,Z -19.008,A -90.000,B 90.000,C 0.000} C_DIS
LIN {X -63.283,Y -11.483,Z -19.087,A -90.000,B 90.000,C 0.000} C_DIS
LIN {X -63.009,Y -11.498,Z -19.204,A -90.000,B 90.000,C 0.000} C_DIS
LIN {X -62.543,Y -11.508,Z -19.398,A -90.000,B 90.000,C 0.000} C_DIS
LIN {X -61.955,Y -11.539,Z -19.648,A -90.000,B 90.000,C 0.000} C_DIS
LIN {X -61.221,Y -11.558,Z -19.948,A -90.000,B 90.000,C 0.000} C_DIS
LIN {X -60.878,Y -11.578,Z -20.092,A -90.000,B 90.000,C 0.000} C_DIS
LIN {X -60.186,Y -11.599,Z -20.377,A -90.000,B 90.000,C 0.000} C_DIS
LIN {X -60.084,Y -11.604,Z -20.417,A -90.000,B 90.000,C 0.000} C_DIS
LIN {X -59.308,Y -11.627,Z -20.717,A -90.000,B 90.000,C 0.000} C_DIS
LIN {X -59.119,Y -11.639,Z -20.780,A -90.000,B 90.000,C 0.000} C_DIS
LIN {X -58.731,Y -11.653,Z -20.903,A -90.000,B 90.000,C 0.000} C_DIS
LIN {X -58.424,Y -11.667,Z -21.003,A -90.000,B 90.000,C 0.000} C_DIS
LIN {X -58.280,Y -11.678,Z -21.044,A -90.000,B 90.000,C 0.000} C_DIS
LIN {X -58.100,Y -11.690,Z -21.098,A -90.000,B 90.000,C 0.000} C_DIS
LIN {X -57.688,Y -11.700,Z -21.210,A -90.000,B 90.000,C 0.000} C_DIS
LIN {X -57.102,Y -11.725,Z -21.376,A -90.000,B 90.000,C 0.000} C_DIS
LIN {X -56.796,Y -11.745,Z -21.453,A -90.000,B 90.000,C 0.000} C_DIS
LIN {X -55.966,Y -11.772,Z -21.643,A -90.000,B 90.000,C 0.000} C_DIS
LIN {X -55.467,Y -11.800,Z -21.744,A -90.000,B 90.000,C 0.000} C_DIS
LIN {X -55.234,Y -11.811,Z -21.793,A -90.000,B 90.000,C 0.000} C_DIS
LIN {X -54.619,Y -11.835,Z -21.917,A -90.000,B 90.000,C 0.000} C_DIS
LIN {X -54.475,Y -11.838,Z -21.943,A -90.000,B 90.000,C 0.000} C_DIS
LIN {X -53.703,Y -11.865,Z -22.073,A -90.000,B 90.000,C 0.000} C_DIS
LIN {X -53.054,Y -11.871,Z -22.198,A -90.000,B 90.000,C 0.000} C_DIS
LIN {X -52.704,Y -11.876,Z -22.258,A -90.000,B 90.000,C 0.000} C_DIS
LIN {X -52.048,Y -11.889,Z -22.377,A -90.000,B 90.000,C 0.000} C_DIS
LIN {X -51.623,Y -11.901,Z -22.452,A -90.000,B 90.000,C 0.000} C_DIS
LIN {X -51.222,Y -11.908,Z -22.517,A -90.000,B 90.000,C 0.000} C_DIS
LIN {X -50.846,Y -11.906,Z -22.585,A -90.000,B 90.000,C 0.000} C_DIS
LIN {X -50.087,Y -11.907,Z -22.723,A -90.000,B 90.000,C 0.000} C_DIS
LIN {X -48.722,Y -11.915,Z -22.964,A -90.000,B 90.000,C 0.000} C_DIS
LIN {X -48.419,Y -11.918,Z -23.018,A -90.000,B 90.000,C 0.000} C_DIS
LIN {X -48.134,Y -11.918,Z -23.073,A -90.000,B 90.000,C 0.000} C_DIS
LIN {X -47.344,Y -11.925,Z -23.220,A -90.000,B 90.000,C 0.000} C_DIS
LIN {X -46.745,Y -11.943,Z -23.320,A -90.000,B 90.000,C 0.000} C_DIS
LIN {X -45.133,Y -12.000,Z -23.610,A -90.000,B 90.000,C 0.000} C_DIS
LIN {X -43.319,Y -12.068,Z -23.946,A -90.000,B 90.000,C 0.000} C_DIS
LIN {X -42.916,Y -12.085,Z -24.025,A -90.000,B 90.000,C 0.000} C_DIS
LIN {X -41.975,Y -12.135,Z -24.203,A -90.000,B 90.000,C 0.000} C_DIS
LIN {X -41.789,Y -12.144,Z -24.238,A -90.000,B 90.000,C 0.000} C_DIS
LIN {X -41.373,Y -12.169,Z -24.313,A -90.000,B 90.000,C 0.000} C_DIS
LIN {X -40.647,Y -12.212,Z -24.457,A -90.000,B 90.000,C 0.000} C_DIS
LIN {X -39.432,Y -12.282,Z -24.696,A -90.000,B 90.000,C 0.000} C_DIS
LIN {X -38.120,Y -12.368,Z -24.972,A -90.000,B 90.000,C 0.000} C_DIS
LIN {X -37.996,Y -12.376,Z -24.996,A -90.000,B 90.000,C 0.000} C_DIS
LIN {X -36.939,Y -12.429,Z -25.219,A -90.000,B 90.000,C 0.000} C_DIS
LIN {X -36.164,Y -12.380,Z -25.254,A -90.000,B 90.000,C 0.000} C_DIS
LIN {X -35.887,Y -12.367,Z -25.267,A -90.000,B 90.000,C 0.000} C_DIS
LIN {X -35.659,Y -12.360,Z -25.283,A -90.000,B 90.000,C 0.000} C_DIS
LIN {X -35.168,Y -12.336,Z -25.304,A -90.000,B 90.000,C 0.000} C_DIS
LIN {X -34.302,Y -12.290,Z -25.338,A -90.000,B 90.000,C 0.000} C_DIS
LIN {X -33.603,Y -12.251,Z -25.368,A -90.000,B 90.000,C 0.000} C_DIS
LIN {X -33.499,Y -12.247,Z -25.375,A -90.000,B 90.000,C 0.000} C_DIS
LIN {X -33.134,Y -12.238,Z -25.407,A -90.000,B 90.000,C 0.000} C_DIS
LIN {X -32.384,Y -12.199,Z -25.484,A -90.000,B 90.000,C 0.000} C_DIS
LIN {X -31.917,Y -12.173,Z -25.530,A -90.000,B 90.000,C 0.000} C_DIS
LIN {X -31.511,Y -12.155,Z -25.575,A -90.000,B 90.000,C 0.000} C_DIS
LIN {X -31.190,Y -12.147,Z -25.617,A -90.000,B 90.000,C 0.000} C_DIS
LIN {X -29.446,Y -12.076,Z -25.869,A -90.000,B 90.000,C 0.000} C_DIS
LIN {X -28.314,Y -12.029,Z -26.037,A -90.000,B 90.000,C 0.000} C_DIS
LIN {X -27.260,Y -11.989,Z -26.193,A -90.000,B 90.000,C 0.000} C_DIS
LIN {X -25.187,Y -11.923,Z -26.530,A -90.000,B 90.000,C 0.000} C_DIS
LIN {X -24.913,Y -11.913,Z -26.573,A -90.000,B 90.000,C 0.000} C_DIS
LIN {X -24.278,Y -11.903,Z -26.684,A -90.000,B 90.000,C 0.000} C_DIS
LIN {X -21.916,Y -11.855,Z -27.111,A -90.000,B 90.000,C 0.000} C_DIS
LIN {X -19.911,Y -11.828,Z -27.523,A -90.000,B 90.000,C 0.000} C_DIS
LIN {X -18.700,Y -11.817,Z -27.777,A -90.000,B 90.000,C 0.000} C_DIS
LIN {X -17.522,Y -11.804,Z -28.030,A -90.000,B 90.000,C 0.000} C_DIS
LIN {X -15.964,Y -11.792,Z -28.372,A -90.000,B 90.000,C 0.000} C_DIS
LIN {X -15.554,Y -11.787,Z -28.460,A -90.000,B 90.000,C 0.000} C_DIS
LIN {X -14.898,Y -11.782,Z -28.599,A -90.000,B 90.000,C 0.000} C_DIS
LIN {X -14.261,Y -11.783,Z -28.736,A -90.000,B 90.000,C 0.000} C_DIS
LIN {X -13.540,Y -11.774,Z -28.887,A -90.000,B 90.000,C 0.000} C_DIS
LIN {X -12.125,Y -11.755,Z -29.188,A -90.000,B 90.000,C 0.000} C_DIS
LIN {X -10.507,Y -11.744,Z -29.516,A -90.000,B 90.000,C 0.000} C_DIS
LIN {X -9.808,Y -11.747,Z -29.665,A -90.000,B 90.000,C 0.000} C_DIS
LIN {X -9.254,Y -11.747,Z -29.785,A -90.000,B 90.000,C 0.000} C_DIS
LIN {X -8.609,Y -11.749,Z -29.914,A -90.000,B 90.000,C 0.000} C_DIS
LIN {X -6.213,Y -11.761,Z -30.398,A -90.000,B 90.000,C 0.000} C_DIS
LIN {X -4.810,Y -11.746,Z -30.671,A -90.000,B 90.000,C 0.000} C_DIS
LIN {X -3.119,Y -11.739,Z -31.008,A -90.000,B 90.000,C 0.000} C_DIS
LIN {X -2.367,Y -11.737,Z -31.147,A -90.000,B 90.000,C 0.000} C_DIS
LIN {X -1.289,Y -11.721,Z -31.337,A -90.000,B 90.000,C 0.000} C_DIS
LIN {X -0.397,Y -11.716,Z -31.483,A -90.000,B 90.000,C 0.000} C_DIS
LIN {X -0.045,Y -11.716,Z -31.543,A -90.000,B 90.000,C 0.000} C_DIS
LIN {X 1.093,Y -11.699,Z -31.735,A -90.000,B 90.000,C 0.000} C_DIS
LIN {X 1.657,Y -11.697,Z -31.821,A -90.000,B 90.000,C 0.000} C_DIS
LIN {X 2.714,Y -11.704,Z -31.992,A -90.000,B 90.000,C 0.000} C_DIS
LIN {X 3.458,Y -11.702,Z -32.126,A -90.000,B 90.000,C 0.000} C_DIS
LIN {X 4.753,Y -11.714,Z -32.339,A -90.000,B 90.000,C 0.000} C_DIS
LIN {X 5.409,Y -11.721,Z -32.449,A -90.000,B 90.000,C 0.000} C_DIS
LIN {X 5.651,Y -11.721,Z -32.497,A -90.000,B 90.000,C 0.000} C_DIS
LIN {X 7.337,Y -11.739,Z -32.812,A -90.000,B 90.000,C 0.000} C_DIS
LIN {X 7.728,Y -11.739,Z -32.882,A -90.000,B 90.000,C 0.000} C_DIS
LIN {X 7.983,Y -11.741,Z -32.930,A -90.000,B 90.000,C 0.000} C_DIS
LIN {X 8.349,Y -11.741,Z -33.012,A -90.000,B 90.000,C 0.000} C_DIS
LIN {X 9.214,Y -11.737,Z -33.212,A -90.000,B 90.000,C 0.000} C_DIS
LIN {X 10.580,Y -11.737,Z -33.533,A -90.000,B 90.000,C 0.000} C_DIS
LIN {X 11.985,Y -11.731,Z -33.882,A -90.000,B 90.000,C 0.000} C_DIS
LIN {X 12.404,Y -11.730,Z -33.986,A -90.000,B 90.000,C 0.000} C_DIS
LIN {X 12.803,Y -11.735,Z -34.079,A -90.000,B 90.000,C 0.000} C_DIS
LIN {X 13.234,Y -11.734,Z -34.180,A -90.000,B 90.000,C 0.000} C_DIS
LIN {X 14.351,Y -11.730,Z -34.443,A -90.000,B 90.000,C 0.000} C_DIS
LIN {X 14.549,Y -11.735,Z -34.482,A -90.000,B 90.000,C 0.000} C_DIS
LIN {X 15.657,Y -11.735,Z -34.681,A -90.000,B 90.000,C 0.000} C_DIS
LIN {X 15.848,Y -11.734,Z -34.715,A -90.000,B 90.000,C 0.000} C_DIS
LIN {X 16.161,Y -11.745,Z -34.754,A -90.000,B 90.000,C 0.000} C_DIS
LIN {X 16.763,Y -11.748,Z -34.794,A -90.000,B 90.000,C 0.000} C_DIS
LIN {X 17.292,Y -11.739,Z -34.822,A -90.000,B 90.000,C 0.000} C_DIS
LIN {X 17.449,Y -11.744,Z -34.820,A -90.000,B 90.000,C 0.000} C_DIS
LIN {X 17.784,Y -11.746,Z -34.813,A -90.000,B 90.000,C 0.000} C_DIS
LIN {X 18.506,Y -11.726,Z -34.781,A -90.000,B 90.000,C 0.000} C_DIS
LIN {X 18.584,Y -11.725,Z -34.778,A -90.000,B 90.000,C 0.000} C_DIS
LIN {X 20.055,Y -11.694,Z -34.660,A -90.000,B 90.000,C 0.000} C_DIS
LIN {X 20.960,Y -11.677,Z -34.593,A -90.000,B 90.000,C 0.000} C_DIS
LIN {X 21.137,Y -11.674,Z -34.580,A -90.000,B 90.000,C 0.000} C_DIS
LIN {X 21.254,Y -11.674,Z -34.574,A -90.000,B 90.000,C 0.000} C_DIS
LIN {X 22.361,Y -11.646,Z -34.550,A -90.000,B 90.000,C 0.000} C_DIS
LIN {X 22.818,Y -11.639,Z -34.545,A -90.000,B 90.000,C 0.000} C_DIS
LIN {X 23.000,Y -11.636,Z -34.547,A -90.000,B 90.000,C 0.000} C_DIS
LIN {X 23.842,Y -11.614,Z -34.572,A -90.000,B 90.000,C 0.000} C_DIS
LIN {X 24.145,Y -11.611,Z -34.583,A -90.000,B 90.000,C 0.000} C_DIS
LIN {X 24.593,Y -11.598,Z -34.616,A -90.000,B 90.000,C 0.000} C_DIS
LIN {X 25.301,Y -11.580,Z -34.676,A -90.000,B 90.000,C 0.000} C_DIS
LIN {X 25.817,Y -11.570,Z -34.722,A -90.000,B 90.000,C 0.000} C_DIS
LIN {X 26.060,Y -11.564,Z -34.749,A -90.000,B 90.000,C 0.000} C_DIS
LIN {X 26.608,Y -11.550,Z -34.812,A -90.000,B 90.000,C 0.000} C_DIS
LIN {X 27.338,Y -11.532,Z -34.909,A -90.000,B 90.000,C 0.000} C_DIS
LIN {X 27.464,Y -11.530,Z -34.926,A -90.000,B 90.000,C 0.000} C_DIS
LIN {X 27.764,Y -11.523,Z -34.973,A -90.000,B 90.000,C 0.000} C_DIS
LIN {X 28.165,Y -11.510,Z -35.039,A -90.000,B 90.000,C 0.000} C_DIS
LIN {X 29.192,Y -11.483,Z -35.199,A -90.000,B 90.000,C 0.000} C_DIS
LIN {X 29.573,Y -11.476,Z -35.260,A -90.000,B 90.000,C 0.000} C_DIS
LIN {X 30.521,Y -11.447,Z -35.432,A -90.000,B 90.000,C 0.000} C_DIS
LIN {X 30.960,Y -11.438,Z -35.507,A -90.000,B 90.000,C 0.000} C_DIS
LIN {X 31.495,Y -11.428,Z -35.599,A -90.000,B 90.000,C 0.000} C_DIS
LIN {X 32.649,Y -11.401,Z -35.825,A -90.000,B 90.000,C 0.000} C_DIS
LIN {X 34.012,Y -11.371,Z -36.112,A -90.000,B 90.000,C 0.000} C_DIS
LIN {X 34.323,Y -11.366,Z -36.178,A -90.000,B 90.000,C 0.000} C_DIS
LIN {X 35.984,Y -11.339,Z -36.579,A -90.000,B 90.000,C 0.000} C_DIS
LIN {X 37.654,Y -11.320,Z -37.028,A -90.000,B 90.000,C 0.000} C_DIS
LIN {X 38.405,Y -11.316,Z -37.240,A -90.000,B 90.000,C 0.000} C_DIS
LIN {X 38.865,Y -11.314,Z -37.377,A -90.000,B 90.000,C 0.000} C_DIS
LIN {X 38.958,Y -11.313,Z -37.408,A -90.000,B 90.000,C 0.000} C_DIS
LIN {X 41.274,Y -11.309,Z -38.102,A -90.000,B 90.000,C 0.000} C_DIS
LIN {X 41.465,Y -11.309,Z -38.161,A -90.000,B 90.000,C 0.000} C_DIS
LIN {X 41.501,Y -11.309,Z -38.173,A -90.000,B 90.000,C 0.000} C_DIS
LIN {X 42.574,Y -11.308,Z -38.529,A -90.000,B 90.000,C 0.000} C_DIS
LIN {X 42.574,Y -60.000,Z -38.529,A -90.000,B 90.000,C 0.000} C_DIS
LIN {X 59.471,Y -60.000,Z -47.736,A -90.000,B 90.000,C 0.000} C_DIS
LIN {X 59.471,Y -11.308,Z -47.736,A -90.000,B 90.000,C 0.000} C_DIS
LIN {X 60.087,Y -11.313,Z -48.081,A -90.000,B 90.000,C 0.000} C_DIS
LIN {X 60.291,Y -11.316,Z -48.199,A -90.000,B 90.000,C 0.000} C_DIS
LIN {X 61.211,Y -11.321,Z -48.724,A -90.000,B 90.000,C 0.000} C_DIS
LIN {X 61.757,Y -11.328,Z -49.001,A -90.000,B 90.000,C 0.000} C_DIS
LIN {X 62.522,Y -11.335,Z -49.396,A -90.000,B 90.000,C 0.000} C_DIS
LIN {X 63.426,Y -11.342,Z -49.858,A -90.000,B 90.000,C 0.000} C_DIS
LIN {X 64.165,Y -11.351,Z -50.222,A -90.000,B 90.000,C 0.000} C_DIS
LIN {X 64.623,Y -11.353,Z -50.451,A -90.000,B 90.000,C 0.000} C_DIS
LIN {X 65.310,Y -11.355,Z -50.799,A -90.000,B 90.000,C 0.000} C_DIS
LIN {X 66.461,Y -11.356,Z -51.391,A -90.000,B 90.000,C 0.000} C_DIS
LIN {X 67.054,Y -11.357,Z -51.704,A -90.000,B 90.000,C 0.000} C_DIS
LIN {X 68.566,Y -11.353,Z -52.539,A -90.000,B 90.000,C 0.000} C_DIS
LIN {X 69.039,Y -11.355,Z -52.799,A -90.000,B 90.000,C 0.000} C_DIS
LIN {X 69.800,Y -11.353,Z -53.244,A -90.000,B 90.000,C 0.000} C_DIS
LIN {X 70.742,Y -11.349,Z -53.798,A -90.000,B 90.000,C 0.000} C_DIS
LIN {X 70.993,Y -11.350,Z -53.946,A -90.000,B 90.000,C 0.000} C_DIS
LIN {X 71.846,Y -11.348,Z -54.477,A -90.000,B 90.000,C 0.000} C_DIS
LIN {X 73.095,Y -11.347,Z -55.249,A -90.000,B 90.000,C 0.000} C_DIS
LIN {X 75.176,Y -11.349,Z -56.605,A -90.000,B 90.000,C 0.000} C_DIS
LIN {X 75.577,Y -11.350,Z -56.873,A -90.000,B 90.000,C 0.000} C_DIS
LIN {X 76.930,Y -11.356,Z -57.810,A -90.000,B 90.000,C 0.000} C_DIS
LIN {X 77.395,Y -11.359,Z -58.140,A -90.000,B 90.000,C 0.000} C_DIS
LIN {X 78.611,Y -11.369,Z -59.053,A -90.000,B 90.000,C 0.000} C_DIS
LIN {X 78.742,Y -11.370,Z -59.154,A -90.000,B 90.000,C 0.000} C_DIS
LIN {X 78.742,Y -60.000,Z -59.154,A -90.000,B 90.000,C 0.000} C_DIS
LIN {X 86.813,Y -60.000,Z -48.200,A -90.000,B 90.000,C 0.000} C_DIS
LIN {X 86.813,Y -11.308,Z -48.200,A -90.000,B 90.000,C 0.000} C_DIS
LIN {X 87.471,Y -11.312,Z -47.534,A -90.000,B 90.000,C 0.000} C_DIS
LIN {X 87.493,Y -11.308,Z -47.512,A -90.000,B 90.000,C 0.000} C_DIS
LIN {X 87.493,Y -60.000,Z -47.512,A -90.000,B 90.000,C 0.000} C_DIS
LIN {X -120.015,Y -60.000,Z -240.907,A -90.000,B 90.000,C 0.000} C_DIS
LIN {X -120.015,Y -11.308,Z -240.907,A -90.000,B 90.000,C 0.000} C_DIS
LIN {X -117.247,Y -11.308,Z -239.026,A -90.000,B 90.000,C 0.000} C_DIS
LIN {X -113.998,Y -11.308,Z -236.843,A -90.000,B 90.000,C 0.000} C_DIS
LIN {X -109.848,Y -11.308,Z -234.062,A -90.000,B 90.000,C 0.000} C_DIS
LIN {X -102.156,Y -11.308,Z -228.976,A -90.000,B 90.000,C 0.000} C_DIS
LIN {X -94.210,Y -11.308,Z -223.811,A -90.000,B 90.000,C 0.000} C_DIS
LIN {X -89.135,Y -11.308,Z -220.577,A -90.000,B 90.000,C 0.000} C_DIS
LIN {X -85.949,Y -11.308,Z -218.553,A -90.000,B 90.000,C 0.000} C_DIS
LIN {X -80.440,Y -11.308,Z -215.129,A -90.000,B 90.000,C 0.000} C_DIS
LIN {X -77.455,Y -11.308,Z -213.297,A -90.000,B 90.000,C 0.000} C_DIS
LIN {X -72.390,Y -11.308,Z -210.226,A -90.000,B 90.000,C 0.000} C_DIS
LIN {X -69.847,Y -11.308,Z -208.690,A -90.000,B 90.000,C 0.000} C_DIS
LIN {X -69.311,Y -11.308,Z -208.368,A -90.000,B 90.000,C 0.000} C_DIS
LIN {X -63.361,Y -11.308,Z -204.780,A -90.000,B 90.000,C 0.000} C_DIS
LIN {X -61.539,Y -11.308,Z -203.695,A -90.000,B 90.000,C 0.000} C_DIS
LIN {X -57.313,Y -11.308,Z -201.114,A -90.000,B 90.000,C 0.000} C_DIS
LIN {X -54.615,Y -11.308,Z -199.489,A -90.000,B 90.000,C 0.000} C_DIS
LIN {X -51.668,Y -11.308,Z -197.646,A -90.000,B 90.000,C 0.000} C_DIS
LIN {X -48.905,Y -11.308,Z -195.899,A -90.000,B 90.000,C 0.000} C_DIS
LIN {X -45.943,Y -11.308,Z -193.965,A -90.000,B 90.000,C 0.000} C_DIS
LIN {X -44.127,Y -11.308,Z -192.765,A -90.000,B 90.000,C 0.000} C_DIS
LIN {X -42.146,Y -11.308,Z -191.410,A -90.000,B 90.000,C 0.000} C_DIS
LIN {X -40.431,Y -11.308,Z -190.223,A -90.000,B 90.000,C 0.000} C_DIS
LIN {X -38.656,Y -11.308,Z -188.957,A -90.000,B 90.000,C 0.000} C_DIS
LIN {X -36.959,Y -11.308,Z -187.730,A -90.000,B 90.000,C 0.000} C_DIS
LIN {X -35.437,Y -11.308,Z -186.596,A -90.000,B 90.000,C 0.000} C_DIS
LIN {X -33.756,Y -11.308,Z -185.358,A -90.000,B 90.000,C 0.000} C_DIS
LIN {X -32.322,Y -11.308,Z -184.241,A -90.000,B 90.000,C 0.000} C_DIS
LIN {X -30.852,Y -11.308,Z -183.112,A -90.000,B 90.000,C 0.000} C_DIS
LIN {X -29.435,Y -11.308,Z -181.946,A -90.000,B 90.000,C 0.000} C_DIS
LIN {X -28.470,Y -11.308,Z -181.159,A -90.000,B 90.000,C 0.000} C_DIS
LIN {X -27.157,Y -11.308,Z -179.996,A -90.000,B 90.000,C 0.000} C_DIS
LIN {X -26.033,Y -11.308,Z -179.009,A -90.000,B 90.000,C 0.000} C_DIS
LIN {X -24.010,Y -11.308,Z -177.055,A -90.000,B 90.000,C 0.000} C_DIS
LIN {X -23.302,Y -11.308,Z -176.288,A -90.000,B 90.000,C 0.000} C_DIS
LIN {X -22.118,Y -11.308,Z -175.018,A -90.000,B 90.000,C 0.000} C_DIS
LIN {X -21.400,Y -11.308,Z -174.130,A -90.000,B 90.000,C 0.000} C_DIS
LIN {X -20.526,Y -11.308,Z -173.070,A -90.000,B 90.000,C 0.000} C_DIS
LIN {X -19.980,Y -11.308,Z -172.290,A -90.000,B 90.000,C 0.000} C_DIS
LIN {X -19.037,Y -11.308,Z -170.976,A -90.000,B 90.000,C 0.000} C_DIS
LIN {X -18.248,Y -11.308,Z -169.695,A -90.000,B 90.000,C 0.000} C_DIS
LIN {X -17.681,Y -11.308,Z -168.755,A -90.000,B 90.000,C 0.000} C_DIS
LIN {X -16.910,Y -11.308,Z -167.280,A -90.000,B 90.000,C 0.000} C_DIS
LIN {X -16.482,Y -11.308,Z -166.456,A -90.000,B 90.000,C 0.000} C_DIS
LIN {X -15.851,Y -11.308,Z -164.959,A -90.000,B 90.000,C 0.000} C_DIS
LIN {X -15.638,Y -11.308,Z -164.459,A -90.000,B 90.000,C 0.000} C_DIS
LIN {X -15.239,Y -11.308,Z -163.088,A -90.000,B 90.000,C 0.000} C_DIS
LIN {X -15.179,Y -11.308,Z -162.892,A -90.000,B 90.000,C 0.000} C_DIS
LIN {X -15.106,Y -11.308,Z -162.060,A -90.000,B 90.000,C 0.000} C_DIS
LIN {X -15.162,Y -11.308,Z -161.680,A -90.000,B 90.000,C 0.000} C_DIS
LIN {X -15.177,Y -11.308,Z -161.560,A -90.000,B 90.000,C 0.000} C_DIS
LIN {X -15.242,Y -11.308,Z -161.392,A -90.000,B 90.000,C 0.000} C_DIS
LIN {X -15.380,Y -11.308,Z -160.998,A -90.000,B 90.000,C 0.000} C_DIS
LIN {X -15.558,Y -11.308,Z -160.681,A -90.000,B 90.000,C 0.000} C_DIS
LIN {X -15.594,Y -11.308,Z -160.606,A -90.000,B 90.000,C 0.000} C_DIS
LIN {X -15.823,Y -11.308,Z -160.137,A -90.000,B 90.000,C 0.000} C_DIS
LIN {X -16.234,Y -11.308,Z -159.462,A -90.000,B 90.000,C 0.000} C_DIS
LIN {X -16.407,Y -11.308,Z -159.131,A -90.000,B 90.000,C 0.000} C_DIS
LIN {X -16.816,Y -11.308,Z -158.560,A -90.000,B 90.000,C 0.000} C_DIS
LIN {X -17.079,Y -11.308,Z -158.163,A -90.000,B 90.000,C 0.000} C_DIS
LIN {X -17.206,Y -11.308,Z -157.959,A -90.000,B 90.000,C 0.000} C_DIS
LIN {X -17.736,Y -11.308,Z -157.326,A -90.000,B 90.000,C 0.000} C_DIS
LIN {X -18.008,Y -11.308,Z -156.997,A -90.000,B 90.000,C 0.000} C_DIS
LIN {X -18.359,Y -11.308,Z -156.535,A -90.000,B 90.000,C 0.000} C_DIS
LIN {X -19.534,Y -11.308,Z -155.295,A -90.000,B 90.000,C 0.000} C_DIS
LIN {X -19.847,Y -11.308,Z -154.953,A -90.000,B 90.000,C 0.000} C_DIS
LIN {X -20.098,Y -11.308,Z -154.670,A -90.000,B 90.000,C 0.000} C_DIS
LIN {X -21.956,Y -11.308,Z -152.876,A -90.000,B 90.000,C 0.000} C_DIS
LIN {X -22.691,Y -11.308,Z -152.133,A -90.000,B 90.000,C 0.000} C_DIS
LIN {X -24.880,Y -11.308,Z -149.981,A -90.000,B 90.000,C 0.000} C_DIS
LIN {X -25.774,Y -11.308,Z -149.070,A -90.000,B 90.000,C 0.000} C_DIS
LIN {X -28.039,Y -11.308,Z -146.647,A -90.000,B 90.000,C 0.000} C_DIS
LIN {X -28.646,Y -11.308,Z -145.992,A -90.000,B 90.000,C 0.000} C_DIS
LIN {X -29.080,Y -11.308,Z -145.514,A -90.000,B 90.000,C 0.000} C_DIS
LIN {X -29.302,Y -11.308,Z -145.261,A -90.000,B 90.000,C 0.000} C_DIS
LIN {X -29.397,Y -11.308,Z -145.146,A -90.000,B 90.000,C 0.000} C_DIS
LIN {X -32.088,Y -11.308,Z -141.796,A -90.000,B 90.000,C 0.000} C_DIS
LIN {X -32.424,Y -11.308,Z -141.370,A -90.000,B 90.000,C 0.000} C_DIS
LIN {X -32.702,Y -11.308,Z -140.971,A -90.000,B 90.000,C 0.000} C_DIS
LIN {X -32.969,Y -11.308,Z -140.540,A -90.000,B 90.000,C 0.000} C_DIS
LIN {X -35.246,Y -11.308,Z -136.931,A -90.000,B 90.000,C 0.000} C_DIS
LIN {X -35.482,Y -11.308,Z -136.505,A -90.000,B 90.000,C 0.000} C_DIS
LIN {X -36.550,Y -11.308,Z -134.456,A -90.000,B 90.000,C 0.000} C_DIS
LIN {X -37.577,Y -11.308,Z -132.478,A -90.000,B 90.000,C 0.000} C_DIS
LIN {X -39.277,Y -11.308,Z -128.695,A -90.000,B 90.000,C 0.000} C_DIS
LIN {X -39.403,Y -11.308,Z -128.407,A -90.000,B 90.000,C 0.000} C_DIS
LIN {X -40.872,Y -11.308,Z -124.859,A -90.000,B 90.000,C 0.000} C_DIS
LIN {X -41.656,Y -11.308,Z -123.002,A -90.000,B 90.000,C 0.000} C_DIS
LIN {X -41.916,Y -11.308,Z -122.444,A -90.000,B 90.000,C 0.000} C_DIS
LIN {X -42.357,Y -11.308,Z -121.509,A -90.000,B 90.000,C 0.000} C_DIS
LIN {X -43.080,Y -11.308,Z -120.253,A -90.000,B 90.000,C 0.000} C_DIS
LIN {X -43.814,Y -11.308,Z -119.207,A -90.000,B 90.000,C 0.000} C_DIS
LIN {X -44.088,Y -11.308,Z -118.815,A -90.000,B 90.000,C 0.000} C_DIS
LIN {X -44.337,Y -11.308,Z -118.497,A -90.000,B 90.000,C 0.000} C_DIS
LIN {X -45.753,Y -11.308,Z -116.718,A -90.000,B 90.000,C 0.000} C_DIS
LIN {X -48.567,Y -11.308,Z -113.314,A -90.000,B 90.000,C 0.000} C_DIS
LIN {X -49.660,Y -11.308,Z -111.991,A -90.000,B 90.000,C 0.000} C_DIS
LIN {X -50.187,Y -11.308,Z -111.359,A -90.000,B 90.000,C 0.000} C_DIS
LIN {X -51.679,Y -11.308,Z -109.496,A -90.000,B 90.000,C 0.000} C_DIS
LIN {X -52.643,Y -11.308,Z -108.298,A -90.000,B 90.000,C 0.000} C_DIS
LIN {X -55.067,Y -11.308,Z -105.083,A -90.000,B 90.000,C 0.000} C_DIS
LIN {X -57.439,Y -11.308,Z -101.855,A -90.000,B 90.000,C 0.000} C_DIS
LIN {X -58.836,Y -11.308,Z -99.974,A -90.000,B 90.000,C 0.000} C_DIS
LIN {X -59.601,Y -11.308,Z -98.941,A -90.000,B 90.000,C 0.000} C_DIS
LIN {X -60.315,Y -11.308,Z -98.039,A -90.000,B 90.000,C 0.000} C_DIS
LIN {X -61.463,Y -11.308,Z -96.581,A -90.000,B 90.000,C 0.000} C_DIS
LIN {X -61.816,Y -11.308,Z -96.122,A -90.000,B 90.000,C 0.000} C_DIS
LIN {X -63.208,Y -11.308,Z -94.561,A -90.000,B 90.000,C 0.000} C_DIS
LIN {X -63.751,Y -11.308,Z -93.930,A -90.000,B 90.000,C 0.000} C_DIS
LIN {X -65.336,Y -11.308,Z -92.364,A -90.000,B 90.000,C 0.000} C_DIS
LIN {X -65.630,Y -11.308,Z -92.059,A -90.000,B 90.000,C 0.000} C_DIS
LIN {X -66.839,Y -11.308,Z -91.004,A -90.000,B 90.000,C 0.000} C_DIS
LIN {X -67.505,Y -11.308,Z -90.394,A -90.000,B 90.000,C 0.000} C_DIS
LIN {X -69.109,Y -11.308,Z -89.139,A -90.000,B 90.000,C 0.000} C_DIS
LIN {X -69.467,Y -11.308,Z -88.848,A -90.000,B 90.000,C 0.000} C_DIS
LIN {X -69.989,Y -11.308,Z -88.463,A -90.000,B 90.000,C 0.000} C_DIS
LIN {X -71.693,Y -11.308,Z -87.240,A -90.000,B 90.000,C 0.000} C_DIS
LIN {X -72.321,Y -11.308,Z -86.810,A -90.000,B 90.000,C 0.000} C_DIS
LIN {X -73.520,Y -11.308,Z -86.005,A -90.000,B 90.000,C 0.000} C_DIS
LIN {X -74.178,Y -11.308,Z -85.579,A -90.000,B 90.000,C 0.000} C_DIS
LIN {X -75.638,Y -11.308,Z -84.644,A -90.000,B 90.000,C 0.000} C_DIS
LIN {X -77.567,Y -11.308,Z -83.441,A -90.000,B 90.000,C 0.000} C_DIS
LIN {X -79.204,Y -11.308,Z -82.416,A -90.000,B 90.000,C 0.000} C_DIS
LIN {X -80.404,Y -11.308,Z -81.632,A -90.000,B 90.000,C 0.000} C_DIS
LIN {X -80.979,Y -11.308,Z -81.244,A -90.000,B 90.000,C 0.000} C_DIS
LIN {X -81.834,Y -11.308,Z -80.650,A -90.000,B 90.000,C 0.000} C_DIS
LIN {X -82.183,Y -11.308,Z -80.399,A -90.000,B 90.000,C 0.000} C_DIS
LIN {X -83.154,Y -11.308,Z -79.660,A -90.000,B 90.000,C 0.000} C_DIS
LIN {X -83.627,Y -11.308,Z -79.285,A -90.000,B 90.000,C 0.000} C_DIS
LIN {X -84.622,Y -11.308,Z -78.444,A -90.000,B 90.000,C 0.000} C_DIS
LIN {X -85.571,Y -11.308,Z -77.608,A -90.000,B 90.000,C 0.000} C_DIS
LIN {X -86.476,Y -11.308,Z -76.828,A -90.000,B 90.000,C 0.000} C_DIS
LIN {X -87.053,Y -11.308,Z -76.372,A -90.000,B 90.000,C 0.000} C_DIS
LIN {X -87.757,Y -11.308,Z -75.901,A -90.000,B 90.000,C 0.000} C_DIS
LIN {X -88.530,Y -11.308,Z -75.455,A -90.000,B 90.000,C 0.000} C_DIS
LIN {X -89.073,Y -11.308,Z -75.180,A -90.000,B 90.000,C 0.000} C_DIS
LIN {X -89.939,Y -11.308,Z -74.790,A -90.000,B 90.000,C 0.000} C_DIS
LIN {X -90.389,Y -11.308,Z -74.607,A -90.000,B 90.000,C 0.000} C_DIS
LIN {X -90.941,Y -11.308,Z -74.405,A -90.000,B 90.000,C 0.000} C_DIS
LIN {X -91.030,Y -11.308,Z -74.374,A -90.000,B 90.000,C 0.000} C_DIS
LIN {X -91.527,Y -11.308,Z -74.217,A -90.000,B 90.000,C 0.000} C_DIS
LIN {X -91.764,Y -11.308,Z -74.153,A -90.000,B 90.000,C 0.000} C_DIS
LIN {X -92.042,Y -11.308,Z -74.095,A -90.000,B 90.000,C 0.000} C_DIS
LIN {X -92.439,Y -11.308,Z -74.029,A -90.000,B 90.000,C 0.000} C_DIS
LIN {X -93.173,Y -11.308,Z -73.932,A -90.000,B 90.000,C 0.000} C_DIS
LIN {X -93.645,Y -11.308,Z -73.895,A -90.000,B 90.000,C 0.000} C_DIS
LIN {X -94.140,Y -11.308,Z -73.831,A -90.000,B 90.000,C 0.000} C_DIS
LIN {X -95.058,Y -11.308,Z -73.746,A -90.000,B 90.000,C 0.000} C_DIS
LIN {X -95.568,Y -11.308,Z -73.674,A -90.000,B 90.000,C 0.000} C_DIS
LIN {X -95.931,Y -11.308,Z -73.620,A -90.000,B 90.000,C 0.000} C_DIS
LIN {X -96.047,Y -11.308,Z -73.610,A -90.000,B 90.000,C 0.000} C_DIS
LIN {X -96.452,Y -11.308,Z -73.561,A -90.000,B 90.000,C 0.000} C_DIS
LIN {X -96.731,Y -11.308,Z -73.508,A -90.000,B 90.000,C 0.000} C_DIS
LIN {X -97.171,Y -11.308,Z -73.404,A -90.000,B 90.000,C 0.000} C_DIS
LIN {X -97.637,Y -11.308,Z -73.327,A -90.000,B 90.000,C 0.000} C_DIS
LIN {X -98.066,Y -11.308,Z -73.225,A -90.000,B 90.000,C 0.000} C_DIS
LIN {X -98.349,Y -11.308,Z -73.133,A -90.000,B 90.000,C 0.000} C_DIS
LIN {X -98.675,Y -11.308,Z -73.014,A -90.000,B 90.000,C 0.000} C_DIS
LIN {X -99.322,Y -11.308,Z -72.816,A -90.000,B 90.000,C 0.000} C_DIS
LIN {X -99.737,Y -11.308,Z -72.666,A -90.000,B 90.000,C 0.000} C_DIS
LIN {X -100.020,Y -11.308,Z -72.539,A -90.000,B 90.000,C 0.000} C_DIS
LIN {X -100.604,Y -11.308,Z -72.228,A -90.000,B 90.000,C 0.000} C_DIS
LIN {X -101.164,Y -11.308,Z -71.956,A -90.000,B 90.000,C 0.000} C_DIS
LIN {X -101.454,Y -11.308,Z -71.812,A -90.000,B 90.000,C 0.000} C_DIS
LIN {X -101.732,Y -11.308,Z -71.653,A -90.000,B 90.000,C 0.000} C_DIS
LIN {X -102.109,Y -11.308,Z -71.397,A -90.000,B 90.000,C 0.000} C_DIS
LIN {X -102.628,Y -11.308,Z -71.037,A -90.000,B 90.000,C 0.000} C_DIS
LIN {X -103.467,Y -11.308,Z -70.406,A -90.000,B 90.000,C 0.000} C_DIS
LIN {X -103.814,Y -11.308,Z -70.110,A -90.000,B 90.000,C 0.000} C_DIS
LIN {X -104.131,Y -11.308,Z -69.836,A -90.000,B 90.000,C 0.000} C_DIS
LIN {X -105.146,Y -11.308,Z -68.890,A -90.000,B 90.000,C 0.000} C_DIS
LIN {X -105.491,Y -11.308,Z -68.525,A -90.000,B 90.000,C 0.000} C_DIS
LIN {X -106.444,Y -11.308,Z -67.489,A -90.000,B 90.000,C 0.000} C_DIS
LIN {X -106.721,Y -11.308,Z -67.174,A -90.000,B 90.000,C 0.000} C_DIS
LIN {X -107.296,Y -11.308,Z -66.468,A -90.000,B 90.000,C 0.000} C_DIS
LIN {X -107.849,Y -11.308,Z -65.768,A -90.000,B 90.000,C 0.000} C_DIS
LIN {X -108.123,Y -11.308,Z -65.404,A -90.000,B 90.000,C 0.000} C_DIS
LIN {X -108.806,Y -11.308,Z -64.465,A -90.000,B 90.000,C 0.000} C_DIS
LIN {X -109.073,Y -11.308,Z -64.084,A -90.000,B 90.000,C 0.000} C_DIS
LIN {X -109.874,Y -11.308,Z -62.803,A -90.000,B 90.000,C 0.000} C_DIS
LIN {X -110.263,Y -11.308,Z -62.153,A -90.000,B 90.000,C 0.000} C_DIS
LIN {X -110.774,Y -11.308,Z -61.179,A -90.000,B 90.000,C 0.000} C_DIS
LIN {X -110.962,Y -11.308,Z -60.763,A -90.000,B 90.000,C 0.000} C_DIS
LIN {X -111.468,Y -11.308,Z -59.492,A -90.000,B 90.000,C 0.000} C_DIS
LIN {X -111.566,Y -11.308,Z -59.220,A -90.000,B 90.000,C 0.000} C_DIS
LIN {X -111.720,Y -11.308,Z -58.779,A -90.000,B 90.000,C 0.000} C_DIS
LIN {X -111.870,Y -11.308,Z -58.274,A -90.000,B 90.000,C 0.000} C_DIS
LIN {X -112.012,Y -11.308,Z -57.796,A -90.000,B 90.000,C 0.000} C_DIS
LIN {X -112.028,Y -11.308,Z -57.728,A -90.000,B 90.000,C 0.000} C_DIS
LIN {X -112.122,Y -11.308,Z -57.282,A -90.000,B 90.000,C 0.000} C_DIS
LIN {X -112.252,Y -11.308,Z -56.574,A -90.000,B 90.000,C 0.000} C_DIS
LIN {X -112.349,Y -11.308,Z -56.108,A -90.000,B 90.000,C 0.000} C_DIS
LIN {X -112.398,Y -11.308,Z -55.844,A -90.000,B 90.000,C 0.000} C_DIS
LIN {X -112.484,Y -11.308,Z -55.453,A -90.000,B 90.000,C 0.000} C_DIS
LIN {X -112.506,Y -11.308,Z -55.365,A -90.000,B 90.000,C 0.000} C_DIS
LIN {X -112.664,Y -11.308,Z -54.669,A -90.000,B 90.000,C 0.000} C_DIS
LIN {X -112.877,Y -11.308,Z -53.941,A -90.000,B 90.000,C 0.000} C_DIS
LIN {X -113.178,Y -11.308,Z -53.024,A -90.000,B 90.000,C 0.000} C_DIS
LIN {X -113.360,Y -11.308,Z -52.461,A -90.000,B 90.000,C 0.000} C_DIS
LIN {X -113.502,Y -11.308,Z -51.915,A -90.000,B 90.000,C 0.000} C_DIS
LIN {X -113.595,Y -11.308,Z -51.469,A -90.000,B 90.000,C 0.000} C_DIS
LIN {X -113.599,Y -11.308,Z -51.445,A -90.000,B 90.000,C 0.000} C_DIS
LIN {X -113.782,Y -11.308,Z -51.057,A -90.000,B 90.000,C 0.000} C_DIS
LIN {X -113.939,Y -11.308,Z -50.706,A -90.000,B 90.000,C 0.000} C_DIS
LIN {X -114.114,Y -11.308,Z -50.263,A -90.000,B 90.000,C 0.000} C_DIS
LIN {X -114.263,Y -11.308,Z -49.868,A -90.000,B 90.000,C 0.000} C_DIS
LIN {X -114.434,Y -11.308,Z -49.373,A -90.000,B 90.000,C 0.000} C_DIS
LIN {X -114.463,Y -11.308,Z -49.286,A -90.000,B 90.000,C 0.000} C_DIS
LIN {X -114.561,Y -11.308,Z -48.902,A -90.000,B 90.000,C 0.000} C_DIS
LIN {X -114.667,Y -11.308,Z -48.448,A -90.000,B 90.000,C 0.000} C_DIS
LIN {X -114.763,Y -11.308,Z -47.970,A -90.000,B 90.000,C 0.000} C_DIS
LIN {X -114.845,Y -11.308,Z -47.135,A -90.000,B 90.000,C 0.000} C_DIS
LIN {X -114.859,Y -11.308,Z -46.765,A -90.000,B 90.000,C 0.000} C_DIS
LIN {X -114.849,Y -11.308,Z -46.324,A -90.000,B 90.000,C 0.000} C_DIS
LIN {X -114.819,Y -11.308,Z -45.943,A -90.000,B 90.000,C 0.000} C_DIS
LIN {X -114.756,Y -11.308,Z -45.485,A -90.000,B 90.000,C 0.000} C_DIS
LIN {X -114.716,Y -11.308,Z -45.273,A -90.000,B 90.000,C 0.000} C_DIS
LIN {X -114.635,Y -11.308,Z -44.907,A -90.000,B 90.000,C 0.000} C_DIS
LIN {X -114.530,Y -11.308,Z -44.496,A -90.000,B 90.000,C 0.000} C_DIS
LIN {X -114.412,Y -11.308,Z -44.152,A -90.000,B 90.000,C 0.000} C_DIS
LIN {X -114.260,Y -11.308,Z -43.756,A -90.000,B 90.000,C 0.000} C_DIS
LIN {X -114.113,Y -11.308,Z -43.434,A -90.000,B 90.000,C 0.000} C_DIS
LIN {X -114.374,Y -11.308,Z -42.849,A -90.000,B 90.000,C 0.000} C_DIS
LIN {X -114.630,Y -11.308,Z -42.238,A -90.000,B 90.000,C 0.000} C_DIS
LIN {X -114.811,Y -11.308,Z -41.776,A -90.000,B 90.000,C 0.000} C_DIS
LIN {X -114.976,Y -11.308,Z -41.322,A -90.000,B 90.000,C 0.000} C_DIS
LIN {X -115.167,Y -11.308,Z -40.736,A -90.000,B 90.000,C 0.000} C_DIS
LIN {X -115.298,Y -11.308,Z -40.319,A -90.000,B 90.000,C 0.000} C_DIS
LIN {X -115.387,Y -11.308,Z -39.952,A -90.000,B 90.000,C 0.000} C_DIS
LIN {X -115.493,Y -11.308,Z -39.497,A -90.000,B 90.000,C 0.000} C_DIS
LIN {X -115.558,Y -11.308,Z -39.145,A -90.000,B 90.000,C 0.000} C_DIS
LIN {X -115.642,Y -11.308,Z -38.476,A -90.000,B 90.000,C 0.000} C_DIS
LIN {X -115.657,Y -11.308,Z -38.346,A -90.000,B 90.000,C 0.000} C_DIS
LIN {X -115.695,Y -11.308,Z -37.922,A -90.000,B 90.000,C 0.000} C_DIS
LIN {X -115.707,Y -11.308,Z -37.619,A -90.000,B 90.000,C 0.000} C_DIS
LIN {X -115.701,Y -11.308,Z -37.164,A -90.000,B 90.000,C 0.000} C_DIS
LIN {X -115.689,Y -11.308,Z -36.861,A -90.000,B 90.000,C 0.000} C_DIS
LIN {X -115.598,Y -11.308,Z -36.120,A -90.000,B 90.000,C 0.000} C_DIS
LIN {X -115.543,Y -11.308,Z -35.841,A -90.000,B 90.000,C 0.000} C_DIS
LIN {X -115.462,Y -11.308,Z -35.496,A -90.000,B 90.000,C 0.000} C_DIS
LIN {X -115.365,Y -11.308,Z -35.122,A -90.000,B 90.000,C 0.000} C_DIS
LIN {X -115.295,Y -11.308,Z -34.867,A -90.000,B 90.000,C 0.000} C_DIS
LIN {X -115.195,Y -11.308,Z -34.568,A -90.000,B 90.000,C 0.000} C_DIS
LIN {X -114.938,Y -11.308,Z -33.899,A -90.000,B 90.000,C 0.000} C_DIS
LIN {X -114.818,Y -11.308,Z -33.640,A -90.000,B 90.000,C 0.000} C_DIS
LIN {X -114.617,Y -11.308,Z -33.252,A -90.000,B 90.000,C 0.000} C_DIS
LIN {X -114.474,Y -11.308,Z -33.002,A -90.000,B 90.000,C 0.000} C_DIS
LIN {X -114.228,Y -11.308,Z -32.635,A -90.000,B 90.000,C 0.000} C_DIS
LIN {X -114.051,Y -11.308,Z -32.390,A -90.000,B 90.000,C 0.000} C_DIS
LIN {X -113.758,Y -11.308,Z -32.046,A -90.000,B 90.000,C 0.000} C_DIS
LIN {X -113.539,Y -11.308,Z -31.810,A -90.000,B 90.000,C 0.000} C_DIS
LIN {X -113.293,Y -11.308,Z -31.570,A -90.000,B 90.000,C 0.000} C_DIS
LIN {X -113.056,Y -11.308,Z -31.334,A -90.000,B 90.000,C 0.000} C_DIS
LIN {X -113.000,Y -11.308,Z -31.271,A -90.000,B 90.000,C 0.000} C_DIS
LIN {X -112.815,Y -11.308,Z -31.022,A -90.000,B 90.000,C 0.000} C_DIS
LIN {X -112.241,Y -11.308,Z -30.183,A -90.000,B 90.000,C 0.000} C_DIS
LIN {X -111.955,Y -11.308,Z -29.790,A -90.000,B 90.000,C 0.000} C_DIS
LIN {X -111.685,Y -11.308,Z -29.462,A -90.000,B 90.000,C 0.000} C_DIS
LIN {X -111.499,Y -11.308,Z -29.230,A -90.000,B 90.000,C 0.000} C_DIS
LIN {X -111.219,Y -11.308,Z -28.912,A -90.000,B 90.000,C 0.000} C_DIS
LIN {X -111.050,Y -11.308,Z -28.728,A -90.000,B 90.000,C 0.000} C_DIS
LIN {X -110.849,Y -11.308,Z -28.504,A -90.000,B 90.000,C 0.000} C_DIS
LIN {X -110.663,Y -11.308,Z -28.321,A -90.000,B 90.000,C 0.000} C_DIS
LIN {X -110.451,Y -11.308,Z -28.107,A -90.000,B 90.000,C 0.000} C_DIS
LIN {X -110.247,Y -11.308,Z -27.923,A -90.000,B 90.000,C 0.000} C_DIS
LIN {X -109.872,Y -11.308,Z -27.584,A -90.000,B 90.000,C 0.000} C_DIS
LIN {X -109.711,Y -11.308,Z -27.439,A -90.000,B 90.000,C 0.000} C_DIS
LIN {X -109.261,Y -11.308,Z -27.066,A -90.000,B 90.000,C 0.000} C_DIS
LIN {X -108.640,Y -11.308,Z -26.630,A -90.000,B 90.000,C 0.000} C_DIS
LIN {X -108.397,Y -11.308,Z -26.462,A -90.000,B 90.000,C 0.000} C_DIS
LIN {X -107.765,Y -11.308,Z -26.114,A -90.000,B 90.000,C 0.000} C_DIS
LIN {X -107.392,Y -11.308,Z -25.913,A -90.000,B 90.000,C 0.000} C_DIS
LIN {X -106.599,Y -11.308,Z -25.577,A -90.000,B 90.000,C 0.000} C_DIS
LIN {X -106.205,Y -11.308,Z -25.421,A -90.000,B 90.000,C 0.000} C_DIS
LIN {X -105.201,Y -11.308,Z -25.096,A -90.000,B 90.000,C 0.000} C_DIS
LIN {X -104.940,Y -11.308,Z -25.026,A -90.000,B 90.000,C 0.000} C_DIS
LIN {X -104.056,Y -11.308,Z -24.780,A -90.000,B 90.000,C 0.000} C_DIS
LIN {X -103.646,Y -11.308,Z -24.672,A -90.000,B 90.000,C 0.000} C_DIS
LIN {X -103.578,Y -11.308,Z -24.656,A -90.000,B 90.000,C 0.000} C_DIS
LIN {X -102.623,Y -11.308,Z -24.407,A -90.000,B 90.000,C 0.000} C_DIS
LIN {X -102.114,Y -11.308,Z -24.255,A -90.000,B 90.000,C 0.000} C_DIS
LIN {X -102.082,Y -11.308,Z -24.172,A -90.000,B 90.000,C 0.000} C_DIS
LIN {X -101.953,Y -11.308,Z -23.898,A -90.000,B 90.000,C 0.000} C_DIS
LIN {X -101.805,Y -11.308,Z -23.594,A -90.000,B 90.000,C 0.000} C_DIS
LIN {X -101.764,Y -11.308,Z -23.515,A -90.000,B 90.000,C 0.000} C_DIS
LIN {X -101.686,Y -11.308,Z -23.350,A -90.000,B 90.000,C 0.000} C_DIS
LIN {X -101.651,Y -11.308,Z -23.280,A -90.000,B 90.000,C 0.000} C_DIS
LIN {X -101.403,Y -11.308,Z -22.847,A -90.000,B 90.000,C 0.000} C_DIS
LIN {X -101.148,Y -11.308,Z -22.489,A -90.000,B 90.000,C 0.000} C_DIS
LIN {X -100.920,Y -11.308,Z -22.175,A -90.000,B 90.000,C 0.000} C_DIS
LIN {X -100.872,Y -11.308,Z -22.115,A -90.000,B 90.000,C 0.000} C_DIS
LIN {X -100.612,Y -11.308,Z -21.826,A -90.000,B 90.000,C 0.000} C_DIS
LIN {X -100.251,Y -11.308,Z -21.462,A -90.000,B 90.000,C 0.000} C_DIS
LIN {X -100.232,Y -11.308,Z -21.445,A -90.000,B 90.000,C 0.000} C_DIS
LIN {X -99.872,Y -11.308,Z -21.155,A -90.000,B 90.000,C 0.000} C_DIS
LIN {X -99.712,Y -11.308,Z -21.043,A -90.000,B 90.000,C 0.000} C_DIS
LIN {X -99.591,Y -11.308,Z -20.962,A -90.000,B 90.000,C 0.000} C_DIS
LIN {X -99.207,Y -11.308,Z -20.716,A -90.000,B 90.000,C 0.000} C_DIS
LIN {X -98.794,Y -11.308,Z -20.510,A -90.000,B 90.000,C 0.000} C_DIS
LIN {X -98.702,Y -11.308,Z -20.470,A -90.000,B 90.000,C 0.000} C_DIS
LIN {X -98.326,Y -11.308,Z -20.319,A -90.000,B 90.000,C 0.000} C_DIS
LIN {X -98.030,Y -11.308,Z -20.178,A -90.000,B 90.000,C 0.000} C_DIS
LIN {X -97.858,Y -11.308,Z -20.064,A -90.000,B 90.000,C 0.000} C_DIS
LIN {X -97.513,Y -11.308,Z -19.778,A -90.000,B 90.000,C 0.000} C_DIS
LIN {X -97.324,Y -11.308,Z -19.606,A -90.000,B 90.000,C 0.000} C_DIS
LIN {X -97.081,Y -11.308,Z -19.391,A -90.000,B 90.000,C 0.000} C_DIS
LIN {X -96.981,Y -11.308,Z -19.304,A -90.000,B 90.000,C 0.000} C_DIS
LIN {X -96.168,Y -11.308,Z -18.577,A -90.000,B 90.000,C 0.000} C_DIS
LIN {X -95.904,Y -11.308,Z -18.363,A -90.000,B 90.000,C 0.000} C_DIS
LIN {X -95.595,Y -11.308,Z -18.119,A -90.000,B 90.000,C 0.000} C_DIS
LIN {X -95.320,Y -11.308,Z -17.921,A -90.000,B 90.000,C 0.000} C_DIS
LIN {X -95.018,Y -11.308,Z -17.728,A -90.000,B 90.000,C 0.000} C_DIS
LIN {X -94.561,Y -11.308,Z -17.465,A -90.000,B 90.000,C 0.000} C_DIS
LIN {X -94.264,Y -11.308,Z -17.296,A -90.000,B 90.000,C 0.000} C_DIS
LIN {X -94.155,Y -11.308,Z -17.242,A -90.000,B 90.000,C 0.000} C_DIS
LIN {X -93.464,Y -11.308,Z -16.945,A -90.000,B 90.000,C 0.000} C_DIS
LIN {X -93.112,Y -11.308,Z -16.802,A -90.000,B 90.000,C 0.000} C_DIS
LIN {X -92.666,Y -11.308,Z -16.663,A -90.000,B 90.000,C 0.000} C_DIS
LIN {X -91.824,Y -11.308,Z -16.427,A -90.000,B 90.000,C 0.000} C_DIS
LIN {X -91.366,Y -11.308,Z -16.337,A -90.000,B 90.000,C 0.000} C_DIS
LIN {X -91.182,Y -11.308,Z -16.306,A -90.000,B 90.000,C 0.000} C_DIS
LIN {X -90.322,Y -11.308,Z -16.169,A -90.000,B 90.000,C 0.000} C_DIS
LIN {X -90.048,Y -11.308,Z -16.145,A -90.000,B 90.000,C 0.000} C_DIS
LIN {X -88.732,Y -11.308,Z -16.069,A -90.000,B 90.000,C 0.000} C_DIS
LIN {X -88.664,Y -11.308,Z -16.070,A -90.000,B 90.000,C 0.000} C_DIS
LIN {X -87.114,Y -11.308,Z -16.144,A -90.000,B 90.000,C 0.000} C_DIS
LIN {X -86.964,Y -11.308,Z -16.167,A -90.000,B 90.000,C 0.000} C_DIS
LIN {X -86.820,Y -11.308,Z -16.007,A -90.000,B 90.000,C 0.000} C_DIS
LIN {X -86.681,Y -11.308,Z -15.870,A -90.000,B 90.000,C 0.000} C_DIS
LIN {X -86.392,Y -11.308,Z -15.607,A -90.000,B 90.000,C 0.000} C_DIS
LIN {X -86.124,Y -11.308,Z -15.385,A -90.000,B 90.000,C 0.000} C_DIS
LIN {X -85.687,Y -11.308,Z -15.053,A -90.000,B 90.000,C 0.000} C_DIS
LIN {X -85.626,Y -11.308,Z -15.010,A -90.000,B 90.000,C 0.000} C_DIS
LIN {X -85.284,Y -11.308,Z -14.785,A -90.000,B 90.000,C 0.000} C_DIS
LIN {X -85.216,Y -11.308,Z -14.745,A -90.000,B 90.000,C 0.000} C_DIS
LIN {X -84.793,Y -11.308,Z -14.527,A -90.000,B 90.000,C 0.000} C_DIS
LIN {X -84.557,Y -11.308,Z -14.419,A -90.000,B 90.000,C 0.000} C_DIS
LIN {X -84.268,Y -11.308,Z -14.277,A -90.000,B 90.000,C 0.000} C_DIS
LIN {X -84.222,Y -11.308,Z -14.257,A -90.000,B 90.000,C 0.000} C_DIS
LIN {X -83.778,Y -11.308,Z -14.085,A -90.000,B 90.000,C 0.000} C_DIS
LIN {X -83.308,Y -11.308,Z -13.958,A -90.000,B 90.000,C 0.000} C_DIS
LIN {X -83.254,Y -11.308,Z -13.944,A -90.000,B 90.000,C 0.000} C_DIS
LIN {X -82.951,Y -11.308,Z -13.855,A -90.000,B 90.000,C 0.000} C_DIS
LIN {X -82.629,Y -11.308,Z -13.767,A -90.000,B 90.000,C 0.000} C_DIS
LIN {X -82.489,Y -11.308,Z -13.732,A -90.000,B 90.000,C 0.000} C_DIS
LIN {X -82.091,Y -11.308,Z -13.666,A -90.000,B 90.000,C 0.000} C_DIS
LIN {X -81.889,Y -11.308,Z -13.637,A -90.000,B 90.000,C 0.000} C_DIS
LIN {X -81.504,Y -11.308,Z -13.560,A -90.000,B 90.000,C 0.000} C_DIS
LIN {X -81.210,Y -11.308,Z -13.512,A -90.000,B 90.000,C 0.000} C_DIS
LIN {X -81.031,Y -11.308,Z -13.488,A -90.000,B 90.000,C 0.000} C_DIS
LIN {X -80.660,Y -11.308,Z -13.452,A -90.000,B 90.000,C 0.000} C_DIS
LIN {X -80.379,Y -11.308,Z -13.429,A -90.000,B 90.000,C 0.000} C_DIS
LIN {X -79.919,Y -11.308,Z -13.373,A -90.000,B 90.000,C 0.000} C_DIS
LIN {X -79.600,Y -11.308,Z -13.355,A -90.000,B 90.000,C 0.000} C_DIS
LIN {X -79.441,Y -11.308,Z -13.349,A -90.000,B 90.000,C 0.000} C_DIS
LIN {X -79.035,Y -11.308,Z -13.341,A -90.000,B 90.000,C 0.000} C_DIS
LIN {X -78.730,Y -11.308,Z -13.341,A -90.000,B 90.000,C 0.000} C_DIS
LIN {X -78.406,Y -11.308,Z -13.335,A -90.000,B 90.000,C 0.000} C_DIS
LIN {X -78.245,Y -11.308,Z -13.340,A -90.000,B 90.000,C 0.000} C_DIS
LIN {X -77.861,Y -11.308,Z -13.359,A -90.000,B 90.000,C 0.000} C_DIS
LIN {X -77.283,Y -11.308,Z -13.405,A -90.000,B 90.000,C 0.000} C_DIS
LIN {X -76.747,Y -11.308,Z -13.481,A -90.000,B 90.000,C 0.000} C_DIS
LIN {X -76.271,Y -11.308,Z -13.564,A -90.000,B 90.000,C 0.000} C_DIS
LIN {X -75.373,Y -11.308,Z -13.764,A -90.000,B 90.000,C 0.000} C_DIS
LIN {X -74.909,Y -11.308,Z -13.895,A -90.000,B 90.000,C 0.000} C_DIS
LIN {X -74.657,Y -11.308,Z -13.970,A -90.000,B 90.000,C 0.000} C_DIS
LIN {X -74.274,Y -11.308,Z -14.120,A -90.000,B 90.000,C 0.000} C_DIS
LIN {X -73.853,Y -11.308,Z -14.291,A -90.000,B 90.000,C 0.000} C_DIS
LIN {X -73.372,Y -11.308,Z -14.469,A -90.000,B 90.000,C 0.000} C_DIS
LIN {X -72.924,Y -11.308,Z -14.648,A -90.000,B 90.000,C 0.000} C_DIS
LIN {X -72.723,Y -11.308,Z -14.739,A -90.000,B 90.000,C 0.000} C_DIS
LIN {X -71.925,Y -11.308,Z -15.066,A -90.000,B 90.000,C 0.000} C_DIS
LIN {X -71.610,Y -11.308,Z -15.201,A -90.000,B 90.000,C 0.000} C_DIS
LIN {X -70.150,Y -11.308,Z -15.859,A -90.000,B 90.000,C 0.000} C_DIS
LIN {X -69.310,Y -11.308,Z -16.246,A -90.000,B 90.000,C 0.000} C_DIS
LIN {X -68.594,Y -11.308,Z -16.584,A -90.000,B 90.000,C 0.000} C_DIS
LIN {X -68.496,Y -11.308,Z -16.633,A -90.000,B 90.000,C 0.000} C_DIS
LIN {X -67.095,Y -11.308,Z -17.301,A -90.000,B 90.000,C 0.000} C_DIS
LIN {X -65.651,Y -11.308,Z -17.975,A -90.000,B 90.000,C 0.000} C_DIS
LIN {X -64.500,Y -11.308,Z -18.488,A -90.000,B 90.000,C 0.000} C_DIS
LIN {X -64.384,Y -11.308,Z -18.544,A -90.000,B 90.000,C 0.000} C_DIS
LIN {X -63.393,Y -11.308,Z -18.965,A -90.000,B 90.000,C 0.000} C_DIS
LIN {X -63.222,Y -11.308,Z -19.042,A -90.000,B 90.000,C 0.000} C_DIS
LIN {X -62.122,Y -11.308,Z -19.490,A -90.000,B 90.000,C 0.000} C_DIS
LIN {X -61.114,Y -11.308,Z -19.891,A -90.000,B 90.000,C 0.000} C_DIS
LIN {X -60.568,Y -11.308,Z -20.097,A -90.000,B 90.000,C 0.000} C_DIS
LIN {X -60.249,Y -11.308,Z -20.225,A -90.000,B 90.000,C 0.000} C_DIS
LIN {X -59.820,Y -11.308,Z -20.368,A -90.000,B 90.000,C 0.000} C_DIS
LIN {X -59.325,Y -11.308,Z -20.544,A -90.000,B 90.000,C 0.000} C_DIS
LIN {X -58.352,Y -11.308,Z -20.835,A -90.000,B 90.000,C 0.000} C_DIS
LIN {X -57.758,Y -11.308,Z -20.970,A -90.000,B 90.000,C 0.000} C_DIS
LIN {X -57.144,Y -11.308,Z -21.103,A -90.000,B 90.000,C 0.000} C_DIS
LIN {X -56.121,Y -11.308,Z -21.134,A -90.000,B 90.000,C 0.000} C_DIS
LIN {X -55.778,Y -11.308,Z -21.139,A -90.000,B 90.000,C 0.000} C_DIS
LIN {X -53.928,Y -11.308,Z -21.291,A -90.000,B 90.000,C 0.000} C_DIS
LIN {X -53.603,Y -11.308,Z -21.319,A -90.000,B 90.000,C 0.000} C_DIS
LIN {X -51.373,Y -11.308,Z -21.569,A -90.000,B 90.000,C 0.000} C_DIS
LIN {X -50.014,Y -11.308,Z -21.732,A -90.000,B 90.000,C 0.000} C_DIS
LIN {X -48.660,Y -11.308,Z -21.912,A -90.000,B 90.000,C 0.000} C_DIS
LIN {X -47.252,Y -11.308,Z -22.104,A -90.000,B 90.000,C 0.000} C_DIS
LIN {X -45.701,Y -11.308,Z -22.285,A -90.000,B 90.000,C 0.000} C_DIS
LIN {X -43.637,Y -11.308,Z -22.594,A -90.000,B 90.000,C 0.000} C_DIS
LIN {X -42.696,Y -11.308,Z -22.761,A -90.000,B 90.000,C 0.000} C_DIS
LIN {X -41.987,Y -11.308,Z -22.867,A -90.000,B 90.000,C 0.000} C_DIS
LIN {X -40.813,Y -11.308,Z -23.058,A -90.000,B 90.000,C 0.000} C_DIS
LIN {X -39.506,Y -11.308,Z -23.229,A -90.000,B 90.000,C 0.000} C_DIS
LIN {X -37.062,Y -11.308,Z -23.638,A -90.000,B 90.000,C 0.000} C_DIS
LIN {X -35.410,Y -11.308,Z -23.968,A -90.000,B 90.000,C 0.000} C_DIS
LIN {X -34.891,Y -11.308,Z -24.062,A -90.000,B 90.000,C 0.000} C_DIS
LIN {X -33.279,Y -11.308,Z -24.359,A -90.000,B 90.000,C 0.000} C_DIS
LIN {X -32.007,Y -11.308,Z -24.600,A -90.000,B 90.000,C 0.000} C_DIS
LIN {X -29.884,Y -11.308,Z -24.997,A -90.000,B 90.000,C 0.000} C_DIS
LIN {X -29.432,Y -11.308,Z -25.085,A -90.000,B 90.000,C 0.000} C_DIS
LIN {X -26.919,Y -11.308,Z -25.581,A -90.000,B 90.000,C 0.000} C_DIS
LIN {X -23.139,Y -11.308,Z -26.398,A -90.000,B 90.000,C 0.000} C_DIS
LIN {X -19.939,Y -11.308,Z -27.112,A -90.000,B 90.000,C 0.000} C_DIS
LIN {X -18.294,Y -11.308,Z -27.481,A -90.000,B 90.000,C 0.000} C_DIS
LIN {X -17.475,Y -11.308,Z -27.661,A -90.000,B 90.000,C 0.000} C_DIS
LIN {X -16.134,Y -11.308,Z -27.963,A -90.000,B 90.000,C 0.000} C_DIS
LIN {X -14.860,Y -11.308,Z -28.239,A -90.000,B 90.000,C 0.000} C_DIS
LIN {X -12.792,Y -11.308,Z -28.684,A -90.000,B 90.000,C 0.000} C_DIS
LIN {X -12.042,Y -11.308,Z -28.851,A -90.000,B 90.000,C 0.000} C_DIS
LIN {X -9.445,Y -11.308,Z -29.390,A -90.000,B 90.000,C 0.000} C_DIS
LIN {X -9.097,Y -11.308,Z -29.468,A -90.000,B 90.000,C 0.000} C_DIS
LIN {X -6.085,Y -11.308,Z -30.114,A -90.000,B 90.000,C 0.000} C_DIS
LIN {X -5.194,Y -11.308,Z -30.287,A -90.000,B 90.000,C 0.000} C_DIS
LIN {X -3.073,Y -11.308,Z -30.715,A -90.000,B 90.000,C 0.000} C_DIS
LIN {X -1.731,Y -11.308,Z -30.966,A -90.000,B 90.000,C 0.000} C_DIS
LIN {X -0.128,Y -11.308,Z -31.235,A -90.000,B 90.000,C 0.000} C_DIS
LIN {X 0.695,Y -11.308,Z -31.382,A -90.000,B 90.000,C 0.000} C_DIS
LIN {X 2.733,Y -11.308,Z -31.699,A -90.000,B 90.000,C 0.000} C_DIS
LIN {X 3.076,Y -11.308,Z -31.762,A -90.000,B 90.000,C 0.000} C_DIS
LIN {X 4.944,Y -11.308,Z -32.056,A -90.000,B 90.000,C 0.000} C_DIS
LIN {X 5.419,Y -11.308,Z -32.139,A -90.000,B 90.000,C 0.000} C_DIS
LIN {X 7.746,Y -11.308,Z -32.602,A -90.000,B 90.000,C 0.000} C_DIS
LIN {X 8.017,Y -11.308,Z -32.648,A -90.000,B 90.000,C 0.000} C_DIS
LIN {X 8.508,Y -11.308,Z -32.752,A -90.000,B 90.000,C 0.000} C_DIS
LIN {X 10.322,Y -11.308,Z -33.179,A -90.000,B 90.000,C 0.000} C_DIS
LIN {X 11.022,Y -11.308,Z -33.338,A -90.000,B 90.000,C 0.000} C_DIS
LIN {X 12.410,Y -11.308,Z -33.687,A -90.000,B 90.000,C 0.000} C_DIS
LIN {X 13.205,Y -11.308,Z -33.863,A -90.000,B 90.000,C 0.000} C_DIS
LIN {X 14.319,Y -11.308,Z -34.127,A -90.000,B 90.000,C 0.000} C_DIS
LIN {X 15.783,Y -11.308,Z -34.391,A -90.000,B 90.000,C 0.000} C_DIS
LIN {X 16.452,Y -11.308,Z -34.457,A -90.000,B 90.000,C 0.000} C_DIS
LIN {X 17.293,Y -11.308,Z -34.511,A -90.000,B 90.000,C 0.000} C_DIS
LIN {X 17.582,Y -11.308,Z -34.523,A -90.000,B 90.000,C 0.000} C_DIS
LIN {X 18.409,Y -11.308,Z -34.500,A -90.000,B 90.000,C 0.000} C_DIS
LIN {X 18.763,Y -11.308,Z -34.504,A -90.000,B 90.000,C 0.000} C_DIS
LIN {X 19.651,Y -11.308,Z -34.439,A -90.000,B 90.000,C 0.000} C_DIS
LIN {X 19.720,Y -11.308,Z -34.437,A -90.000,B 90.000,C 0.000} C_DIS
LIN {X 20.554,Y -11.308,Z -34.381,A -90.000,B 90.000,C 0.000} C_DIS
LIN {X 21.002,Y -11.308,Z -34.353,A -90.000,B 90.000,C 0.000} C_DIS
LIN {X 21.436,Y -11.308,Z -34.344,A -90.000,B 90.000,C 0.000} C_DIS
LIN {X 21.717,Y -11.308,Z -34.343,A -90.000,B 90.000,C 0.000} C_DIS
LIN {X 22.696,Y -11.308,Z -34.346,A -90.000,B 90.000,C 0.000} C_DIS
LIN {X 22.804,Y -11.308,Z -34.349,A -90.000,B 90.000,C 0.000} C_DIS
LIN {X 24.249,Y -11.308,Z -34.437,A -90.000,B 90.000,C 0.000} C_DIS
LIN {X 25.035,Y -11.308,Z -34.513,A -90.000,B 90.000,C 0.000} C_DIS
LIN {X 25.608,Y -11.308,Z -34.578,A -90.000,B 90.000,C 0.000} C_DIS
LIN {X 26.218,Y -11.308,Z -34.657,A -90.000,B 90.000,C 0.000} C_DIS
LIN {X 27.256,Y -11.308,Z -34.806,A -90.000,B 90.000,C 0.000} C_DIS
LIN {X 27.782,Y -11.308,Z -34.893,A -90.000,B 90.000,C 0.000} C_DIS
LIN {X 28.466,Y -11.308,Z -35.015,A -90.000,B 90.000,C 0.000} C_DIS
LIN {X 29.592,Y -11.308,Z -35.203,A -90.000,B 90.000,C 0.000} C_DIS
LIN {X 30.905,Y -11.308,Z -35.456,A -90.000,B 90.000,C 0.000} C_DIS
LIN {X 31.482,Y -11.308,Z -35.558,A -90.000,B 90.000,C 0.000} C_DIS
LIN {X 32.312,Y -11.308,Z -35.726,A -90.000,B 90.000,C 0.000} C_DIS
LIN {X 33.611,Y -11.308,Z -36.010,A -90.000,B 90.000,C 0.000} C_DIS
LIN {X 34.121,Y -11.308,Z -36.119,A -90.000,B 90.000,C 0.000} C_DIS
LIN {X 35.926,Y -11.308,Z -36.562,A -90.000,B 90.000,C 0.000} C_DIS
LIN {X 37.617,Y -11.308,Z -37.018,A -90.000,B 90.000,C 0.000} C_DIS
LIN {X 38.406,Y -11.308,Z -37.240,A -90.000,B 90.000,C 0.000} C_DIS
LIN {X 38.866,Y -11.308,Z -37.377,A -90.000,B 90.000,C 0.000} C_DIS
LIN {X 38.960,Y -11.308,Z -37.409,A -90.000,B 90.000,C 0.000} C_DIS
LIN {X 41.465,Y -11.308,Z -38.161,A -90.000,B 90.000,C 0.000} C_DIS
LIN {X 42.646,Y -11.308,Z -38.553,A -90.000,B 90.000,C 0.000} C_DIS
LIN {X 43.564,Y -11.308,Z -38.820,A -90.000,B 90.000,C 0.000} C_DIS
LIN {X 43.897,Y -11.308,Z -38.920,A -90.000,B 90.000,C 0.000} C_DIS
LIN {X 46.609,Y -11.308,Z -39.873,A -90.000,B 90.000,C 0.000} C_DIS
LIN {X 47.060,Y -11.308,Z -40.059,A -90.000,B 90.000,C 0.000} C_DIS
LIN {X 47.136,Y -11.308,Z -40.092,A -90.000,B 90.000,C 0.000} C_DIS
LIN {X 49.496,Y -11.308,Z -41.120,A -90.000,B 90.000,C 0.000} C_DIS
LIN {X 49.806,Y -11.308,Z -41.280,A -90.000,B 90.000,C 0.000} C_DIS
LIN {X 52.095,Y -11.308,Z -42.494,A -90.000,B 90.000,C 0.000} C_DIS
LIN {X 52.501,Y -11.308,Z -42.714,A -90.000,B 90.000,C 0.000} C_DIS
LIN {X 52.707,Y -11.308,Z -42.829,A -90.000,B 90.000,C 0.000} C_DIS
LIN {X 55.125,Y -11.308,Z -44.354,A -90.000,B 90.000,C 0.000} C_DIS
LIN {X 55.508,Y -11.308,Z -44.614,A -90.000,B 90.000,C 0.000} C_DIS
LIN {X 57.720,Y -11.308,Z -46.256,A -90.000,B 90.000,C 0.000} C_DIS
LIN {X 59.471,Y -11.308,Z -47.736,A -90.000,B 90.000,C 0.000} C_DIS
LIN {X 60.053,Y -11.308,Z -48.062,A -90.000,B 90.000,C 0.000} C_DIS
LIN {X 61.195,Y -11.308,Z -48.713,A -90.000,B 90.000,C 0.000} C_DIS
LIN {X 61.754,Y -11.308,Z -48.995,A -90.000,B 90.000,C 0.000} C_DIS
LIN {X 62.928,Y -11.308,Z -49.598,A -90.000,B 90.000,C 0.000} C_DIS
LIN {X 63.427,Y -11.308,Z -49.851,A -90.000,B 90.000,C 0.000} C_DIS
LIN {X 64.141,Y -11.308,Z -50.200,A -90.000,B 90.000,C 0.000} C_DIS
LIN {X 64.615,Y -11.308,Z -50.436,A -90.000,B 90.000,C 0.000} C_DIS
LIN {X 65.286,Y -11.308,Z -50.775,A -90.000,B 90.000,C 0.000} C_DIS
LIN {X 66.388,Y -11.308,Z -51.340,A -90.000,B 90.000,C 0.000} C_DIS
LIN {X 67.088,Y -11.308,Z -51.710,A -90.000,B 90.000,C 0.000} C_DIS
LIN {X 68.509,Y -11.308,Z -52.496,A -90.000,B 90.000,C 0.000} C_DIS
LIN {X 69.058,Y -11.308,Z -52.798,A -90.000,B 90.000,C 0.000} C_DIS
LIN {X 69.605,Y -11.308,Z -53.118,A -90.000,B 90.000,C 0.000} C_DIS
LIN {X 71.002,Y -11.308,Z -53.942,A -90.000,B 90.000,C 0.000} C_DIS
LIN {X 71.612,Y -11.308,Z -54.322,A -90.000,B 90.000,C 0.000} C_DIS
LIN {X 73.103,Y -11.308,Z -55.245,A -90.000,B 90.000,C 0.000} C_DIS
LIN {X 75.184,Y -11.308,Z -56.601,A -90.000,B 90.000,C 0.000} C_DIS
LIN {X 75.586,Y -11.308,Z -56.868,A -90.000,B 90.000,C 0.000} C_DIS
LIN {X 76.919,Y -11.308,Z -57.789,A -90.000,B 90.000,C 0.000} C_DIS
LIN {X 77.406,Y -11.308,Z -58.133,A -90.000,B 90.000,C 0.000} C_DIS
LIN {X 78.697,Y -11.308,Z -59.099,A -90.000,B 90.000,C 0.000} C_DIS
LIN {X 78.745,Y -11.308,Z -59.137,A -90.000,B 90.000,C 0.000} C_DIS
LIN {X 79.009,Y -11.329,Z -59.342,A -90.000,B 90.000,C 0.000} C_DIS
LIN {X 79.248,Y -11.309,Z -59.525,A -90.000,B 90.000,C 0.000} C_DIS
LIN {X 79.543,Y -11.308,Z -59.748,A -90.000,B 90.000,C 0.000} C_DIS
LIN {X 79.544,Y -17.837,Z -59.749,A -90.000,B 90.000,C 0.000} C_DIS
LIN {X 79.548,Y -17.904,Z -59.751,A -90.000,B 90.000,C 0.000} C_DIS
LIN {X 79.560,Y -18.104,Z -59.760,A -90.000,B 90.000,C 0.000} C_DIS
LIN {X 79.607,Y -18.560,Z -59.795,A -90.000,B 90.000,C 0.000} C_DIS
LIN {X 79.652,Y -18.787,Z -59.828,A -90.000,B 90.000,C 0.000} C_DIS
LIN {X 79.739,Y -19.095,Z -59.892,A -90.000,B 90.000,C 0.000} C_DIS
LIN {X 79.821,Y -19.318,Z -59.949,A -90.000,B 90.000,C 0.000} C_DIS
LIN {X 79.898,Y -19.461,Z -60.002,A -90.000,B 90.000,C 0.000} C_DIS
LIN {X 80.037,Y -19.640,Z -60.093,A -90.000,B 90.000,C 0.000} C_DIS
LIN {X 80.173,Y -19.802,Z -60.172,A -90.000,B 90.000,C 0.000} C_DIS
LIN {X 80.180,Y -25.675,Z -60.176,A -90.000,B 90.000,C 0.000} C_DIS
LIN {X 80.186,Y -25.840,Z -60.179,A -90.000,B 90.000,C 0.000} C_DIS
LIN {X 80.213,Y -26.147,Z -60.193,A -90.000,B 90.000,C 0.000} C_DIS
LIN {X 80.310,Y -26.786,Z -60.235,A -90.000,B 90.000,C 0.000} C_DIS
LIN {X 80.353,Y -27.033,Z -60.249,A -90.000,B 90.000,C 0.000} C_DIS
LIN {X 80.393,Y -27.209,Z -60.258,A -90.000,B 90.000,C 0.000} C_DIS
LIN {X 80.446,Y -27.400,Z -60.263,A -90.000,B 90.000,C 0.000} C_DIS
LIN {X 80.478,Y -27.495,Z -60.261,A -90.000,B 90.000,C 0.000} C_DIS
LIN {X 80.507,Y -27.572,Z -60.254,A -90.000,B 90.000,C 0.000} C_DIS
LIN {X 80.534,Y -27.633,Z -60.243,A -90.000,B 90.000,C 0.000} C_DIS
LIN {X 80.558,Y -27.682,Z -60.227,A -90.000,B 90.000,C 0.000} C_DIS
LIN {X 80.580,Y -27.719,Z -60.207,A -90.000,B 90.000,C 0.000} C_DIS
LIN {X 80.599,Y -27.746,Z -60.182,A -90.000,B 90.000,C 0.000} C_DIS
LIN {X 80.609,Y -27.756,Z -60.168,A -90.000,B 90.000,C 0.000} C_DIS
LIN {X 80.626,Y -27.770,Z -60.137,A -90.000,B 90.000,C 0.000} C_DIS
LIN {X 80.641,Y -27.777,Z -60.102,A -90.000,B 90.000,C 0.000} C_DIS
LIN {X 80.655,Y -27.776,Z -60.062,A -90.000,B 90.000,C 0.000} C_DIS
LIN {X 80.668,Y -27.768,Z -60.018,A -90.000,B 90.000,C 0.000} C_DIS
LIN {X 80.680,Y -27.754,Z -59.970,A -90.000,B 90.000,C 0.000} C_DIS
LIN {X 80.691,Y -27.734,Z -59.917,A -90.000,B 90.000,C 0.000} C_DIS
LIN {X 80.701,Y -27.708,Z -59.861,A -90.000,B 90.000,C 0.000} C_DIS
LIN {X 80.711,Y -27.674,Z -59.800,A -90.000,B 90.000,C 0.000} C_DIS
LIN {X 80.729,Y -27.580,Z -59.667,A -90.000,B 90.000,C 0.000} C_DIS
LIN {X 80.748,Y -27.449,Z -59.518,A -90.000,B 90.000,C 0.000} C_DIS
LIN {X 80.768,Y -27.289,Z -59.353,A -90.000,B 90.000,C 0.000} C_DIS
LIN {X 80.791,Y -27.155,Z -59.174,A -90.000,B 90.000,C 0.000} C_DIS
LIN {X 80.835,Y -26.977,Z -58.876,A -90.000,B 90.000,C 0.000} C_DIS
LIN {X 80.894,Y -26.777,Z -58.546,A -90.000,B 90.000,C 0.000} C_DIS
LIN {X 80.944,Y -26.636,Z -58.308,A -90.000,B 90.000,C 0.000} C_DIS
LIN {X 81.005,Y -26.495,Z -58.057,A -90.000,B 90.000,C 0.000} C_DIS
LIN {X 81.039,Y -26.427,Z -57.926,A -90.000,B 90.000,C 0.000} C_DIS
LIN {X 81.077,Y -26.363,Z -57.792,A -90.000,B 90.000,C 0.000} C_DIS
LIN {X 81.118,Y -26.306,Z -57.655,A -90.000,B 90.000,C 0.000} C_DIS
LIN {X 81.162,Y -26.259,Z -57.514,A -90.000,B 90.000,C 0.000} C_DIS
LIN {X 81.210,Y -26.224,Z -57.371,A -90.000,B 90.000,C 0.000} C_DIS
LIN {X 81.262,Y -26.171,Z -57.224,A -90.000,B 90.000,C 0.000} C_DIS
LIN {X 81.378,Y -26.000,Z -56.921,A -90.000,B 90.000,C 0.000} C_DIS
LIN {X 81.442,Y -25.932,Z -56.765,A -90.000,B 90.000,C 0.000} C_DIS
LIN {X 81.512,Y -11.308,Z -56.605,A -90.000,B 90.000,C 0.000} C_DIS
LIN {X 81.700,Y -11.308,Z -56.182,A -90.000,B 90.000,C 0.000} C_DIS
LIN {X 82.134,Y -11.308,Z -55.110,A -90.000,B 90.000,C 0.000} C_DIS
LIN {X 82.335,Y -11.308,Z -54.666,A -90.000,B 90.000,C 0.000} C_DIS
LIN {X 83.331,Y -11.308,Z -52.811,A -90.000,B 90.000,C 0.000} C_DIS
LIN {X 83.577,Y -11.308,Z -52.389,A -90.000,B 90.000,C 0.000} C_DIS
LIN {X 84.737,Y -11.308,Z -50.685,A -90.000,B 90.000,C 0.000} C_DIS
LIN {X 85.025,Y -11.308,Z -50.291,A -90.000,B 90.000,C 0.000} C_DIS
LIN {X 86.337,Y -11.308,Z -48.714,A -90.000,B 90.000,C 0.000} C_DIS
LIN {X 86.664,Y -11.308,Z -48.352,A -90.000,B 90.000,C 0.000} C_DIS
LIN {X 88.117,Y -11.308,Z -46.880,A -90.000,B 90.000,C 0.000} C_DIS
LIN {X 88.479,Y -11.308,Z -46.553,A -90.000,B 90.000,C 0.000} C_DIS
LIN {X 90.061,Y -11.308,Z -45.164,A -90.000,B 90.000,C 0.000} C_DIS
LIN {X 91.716,Y -11.308,Z -43.876,A -90.000,B 90.000,C 0.000} C_DIS
LIN {X 92.110,Y -11.308,Z -43.588,A -90.000,B 90.000,C 0.000} C_DIS
LIN {X 93.780,Y -11.308,Z -42.419,A -90.000,B 90.000,C 0.000} C_DIS
LIN {X 95.417,Y -11.308,Z -41.383,A -90.000,B 90.000,C 0.000} C_DIS
LIN {X 95.838,Y -11.308,Z -41.136,A -90.000,B 90.000,C 0.000} C_DIS
LIN {X 97.376,Y -11.308,Z -40.260,A -90.000,B 90.000,C 0.000} C_DIS
LIN {X 98.805,Y -11.308,Z -39.523,A -90.000,B 90.000,C 0.000} C_DIS
LIN {X 98.814,Y -11.308,Z -39.518,A -90.000,B 90.000,C 0.000} C_DIS
LIN {X 98.814,Y -60.000,Z -39.518,A -90.000,B 90.000,C 0.000} C_DIS
LIN {X 101.451,Y -60.000,Z -88.669,A -90.000,B 90.000,C 0.000} C_DIS
LIN {X 101.451,Y -11.308,Z -88.669,A -90.000,B 90.000,C 0.000} C_DIS
LIN {X 101.949,Y -11.308,Z -89.576,A -90.000,B 90.000,C 0.000} C_DIS
LIN {X 102.113,Y -11.308,Z -89.881,A -90.000,B 90.000,C 0.000} C_DIS
LIN {X 102.684,Y -11.308,Z -91.081,A -90.000,B 90.000,C 0.000} C_DIS
LIN {X 102.855,Y -11.308,Z -91.503,A -90.000,B 90.000,C 0.000} C_DIS
LIN {X 103.300,Y -11.308,Z -92.636,A -90.000,B 90.000,C 0.000} C_DIS
LIN {X 103.650,Y -11.308,Z -93.740,A -90.000,B 90.000,C 0.000} C_DIS
LIN {X 103.774,Y -11.308,Z -94.179,A -90.000,B 90.000,C 0.000} C_DIS
LIN {X 104.062,Y -11.308,Z -95.289,A -90.000,B 90.000,C 0.000} C_DIS
LIN {X 104.322,Y -11.308,Z -96.439,A -90.000,B 90.000,C 0.000} C_DIS
LIN {X 104.583,Y -11.308,Z -97.659,A -90.000,B 90.000,C 0.000} C_DIS
LIN {X 104.859,Y -11.308,Z -99.015,A -90.000,B 90.000,C 0.000} C_DIS
LIN {X 105.163,Y -11.308,Z -100.577,A -90.000,B 90.000,C 0.000} C_DIS
LIN {X 105.392,Y -11.308,Z -101.811,A -90.000,B 90.000,C 0.000} C_DIS
LIN {X 105.629,Y -11.308,Z -103.057,A -90.000,B 90.000,C 0.000} C_DIS
LIN {X 105.904,Y -11.308,Z -104.606,A -90.000,B 90.000,C 0.000} C_DIS
LIN {X 106.013,Y -11.308,Z -105.199,A -90.000,B 90.000,C 0.000} C_DIS
LIN {X 106.329,Y -11.308,Z -107.071,A -90.000,B 90.000,C 0.000} C_DIS
LIN {X 106.630,Y -11.308,Z -108.840,A -90.000,B 90.000,C 0.000} C_DIS
LIN {X 107.034,Y -11.308,Z -111.403,A -90.000,B 90.000,C 0.000} C_DIS
LIN {X 107.253,Y -11.308,Z -112.921,A -90.000,B 90.000,C 0.000} C_DIS
LIN {X 107.485,Y -11.308,Z -114.743,A -90.000,B 90.000,C 0.000} C_DIS
LIN {X 107.620,Y -11.308,Z -115.728,A -90.000,B 90.000,C 0.000} C_DIS
LIN {X 107.854,Y -11.308,Z -117.831,A -90.000,B 90.000,C 0.000} C_DIS
LIN {X 107.937,Y -11.308,Z -118.530,A -90.000,B 90.000,C 0.000} C_DIS
LIN {X 108.166,Y -11.308,Z -120.902,A -90.000,B 90.000,C 0.000} C_DIS
LIN {X 108.205,Y -11.308,Z -121.286,A -90.000,B 90.000,C 0.000} C_DIS
LIN {X 108.419,Y -11.308,Z -123.869,A -90.000,B 90.000,C 0.000} C_DIS
LIN {X 108.427,Y -11.308,Z -123.962,A -90.000,B 90.000,C 0.000} C_DIS
LIN {X 108.608,Y -11.308,Z -126.584,A -90.000,B 90.000,C 0.000} C_DIS
LIN {X 108.766,Y -11.308,Z -129.534,A -90.000,B 90.000,C 0.000} C_DIS
LIN {X 108.861,Y -11.308,Z -132.195,A -90.000,B 90.000,C 0.000} C_DIS
LIN {X 108.916,Y -11.308,Z -135.052,A -90.000,B 90.000,C 0.000} C_DIS
LIN {X 108.928,Y -11.308,Z -138.206,A -90.000,B 90.000,C 0.000} C_DIS
LIN {X 108.885,Y -11.308,Z -141.737,A -90.000,B 90.000,C 0.000} C_DIS
LIN {X 108.778,Y -11.308,Z -145.329,A -90.000,B 90.000,C 0.000} C_DIS
LIN {X 108.594,Y -11.308,Z -149.065,A -90.000,B 90.000,C 0.000} C_DIS
LIN {X 108.320,Y -11.308,Z -152.893,A -90.000,B 90.000,C 0.000} C_DIS
LIN {X 107.943,Y -11.308,Z -157.194,A -90.000,B 90.000,C 0.000} C_DIS
LIN {X 107.572,Y -11.308,Z -160.881,A -90.000,B 90.000,C 0.000} C_DIS
LIN {X 107.179,Y -11.308,Z -164.520,A -90.000,B 90.000,C 0.000} C_DIS
LIN {X 107.093,Y -11.308,Z -165.244,A -90.000,B 90.000,C 0.000} C_DIS
LIN {X 106.733,Y -11.308,Z -168.497,A -90.000,B 90.000,C 0.000} C_DIS
LIN {X 106.328,Y -11.308,Z -172.043,A -90.000,B 90.000,C 0.000} C_DIS
LIN {X 105.927,Y -11.308,Z -175.408,A -90.000,B 90.000,C 0.000} C_DIS
LIN {X 105.529,Y -11.308,Z -178.549,A -90.000,B 90.000,C 0.000} C_DIS
LIN {X 105.135,Y -11.308,Z -181.425,A -90.000,B 90.000,C 0.000} C_DIS
LIN {X 105.068,Y -11.308,Z -181.895,A -90.000,B 90.000,C 0.000} C_DIS
LIN {X 104.680,Y -11.308,Z -184.538,A -90.000,B 90.000,C 0.000} C_DIS
LIN {X 104.294,Y -11.308,Z -187.036,A -90.000,B 90.000,C 0.000} C_DIS
LIN {X 103.795,Y -11.308,Z -190.158,A -90.000,B 90.000,C 0.000} C_DIS
LIN {X 103.526,Y -11.308,Z -191.822,A -90.000,B 90.000,C 0.000} C_DIS
LIN {X 103.094,Y -11.308,Z -194.399,A -90.000,B 90.000,C 0.000} C_DIS
LIN {X 102.574,Y -11.308,Z -197.372,A -90.000,B 90.000,C 0.000} C_DIS
LIN {X 101.920,Y -11.308,Z -200.958,A -90.000,B 90.000,C 0.000} C_DIS
LIN {X 101.089,Y -11.308,Z -205.369,A -90.000,B 90.000,C 0.000} C_DIS
LIN {X 100.090,Y -11.308,Z -210.392,A -90.000,B 90.000,C 0.000} C_DIS
LIN {X 99.303,Y -11.308,Z -214.075,A -90.000,B 90.000,C 0.000} C_DIS
LIN {X 98.933,Y -11.308,Z -215.816,A -90.000,B 90.000,C 0.000} C_DIS
LIN {X 98.134,Y -11.308,Z -219.236,A -90.000,B 90.000,C 0.000} C_DIS
LIN {X 97.628,Y -11.308,Z -221.431,A -90.000,B 90.000,C 0.000} C_DIS
LIN {X 96.985,Y -11.308,Z -223.951,A -90.000,B 90.000,C 0.000} C_DIS
LIN {X 96.161,Y -11.308,Z -227.123,A -90.000,B 90.000,C 0.000} C_DIS
LIN {X 96.081,Y -11.308,Z -227.416,A -90.000,B 90.000,C 0.000} C_DIS
LIN {X 95.237,Y -11.308,Z -230.420,A -90.000,B 90.000,C 0.000} C_DIS
LIN {X 94.466,Y -11.308,Z -233.112,A -90.000,B 90.000,C 0.000} C_DIS
LIN {X 93.366,Y -11.308,Z -236.704,A -90.000,B 90.000,C 0.000} C_DIS
LIN {X 92.640,Y -11.308,Z -239.023,A -90.000,B 90.000,C 0.000} C_DIS
LIN {X 91.142,Y -11.308,Z -243.561,A -90.000,B 90.000,C 0.000} C_DIS
LIN {X 91.142,Y -60.000,Z -243.561,A -90.000,B 90.000,C 0.000} C_DIS
LIN {X 102.464,Y -60.000,Z -88.724,A -90.000,B 90.000,C 0.000} C_DIS
LIN {X 102.464,Y -9.504,Z -88.724,A -90.000,B 90.000,C 0.000} C_DIS
LIN {X 102.864,Y -9.499,Z -89.477,A -90.000,B 90.000,C 0.000} C_DIS
LIN {X 102.986,Y -9.503,Z -89.714,A -90.000,B 90.000,C 0.000} C_DIS
LIN {X 103.166,Y -9.502,Z -90.095,A -90.000,B 90.000,C 0.000} C_DIS
LIN {X 103.457,Y -9.499,Z -90.723,A -90.000,B 90.000,C 0.000} C_DIS
LIN {X 103.552,Y -9.503,Z -90.932,A -90.000,B 90.000,C 0.000} C_DIS
LIN {X 103.849,Y -9.501,Z -91.693,A -90.000,B 90.000,C 0.000} C_DIS
LIN {X 104.089,Y -9.500,Z -92.308,A -90.000,B 90.000,C 0.000} C_DIS
LIN {X 104.161,Y -9.504,Z -92.498,A -90.000,B 90.000,C 0.000} C_DIS
LIN {X 104.392,Y -9.504,Z -93.226,A -90.000,B 90.000,C 0.000} C_DIS
LIN {X 104.508,Y -9.506,Z -93.587,A -90.000,B 90.000,C 0.000} C_DIS
LIN {X 104.632,Y -9.506,Z -94.038,A -90.000,B 90.000,C 0.000} C_DIS
LIN {X 104.861,Y -9.507,Z -94.909,A -90.000,B 90.000,C 0.000} C_DIS
LIN {X 104.920,Y -9.508,Z -95.131,A -90.000,B 90.000,C 0.000} C_DIS
LIN {X 105.132,Y -9.510,Z -96.051,A -90.000,B 90.000,C 0.000} C_DIS
LIN {X 105.184,Y -9.511,Z -96.274,A -90.000,B 90.000,C 0.000} C_DIS
LIN {X 105.456,Y -9.515,Z -97.507,A -90.000,B 90.000,C 0.000} C_DIS
LIN {X 105.747,Y -9.520,Z -98.886,A -90.000,B 90.000,C 0.000} C_DIS
LIN {X 106.058,Y -9.527,Z -100.411,A -90.000,B 90.000,C 0.000} C_DIS
LIN {X 106.316,Y -9.534,Z -101.732,A -90.000,B 90.000,C 0.000} C_DIS
LIN {X 106.562,Y -9.542,Z -102.943,A -90.000,B 90.000,C 0.000} C_DIS
LIN {X 106.858,Y -9.552,Z -104.498,A -90.000,B 90.000,C 0.000} C_DIS
LIN {X 106.973,Y -9.557,Z -105.091,A -90.000,B 90.000,C 0.000} C_DIS
LIN {X 107.408,Y -9.574,Z -107.473,A -90.000,B 90.000,C 0.000} C_DIS
LIN {X 107.620,Y -9.577,Z -108.684,A -90.000,B 90.000,C 0.000} C_DIS
LIN {X 107.812,Y -9.585,Z -109.815,A -90.000,B 90.000,C 0.000} C_DIS
LIN {X 108.024,Y -9.593,Z -111.078,A -90.000,B 90.000,C 0.000} C_DIS
LIN {X 108.185,Y -9.600,Z -112.099,A -90.000,B 90.000,C 0.000} C_DIS
LIN {X 108.293,Y -9.605,Z -112.790,A -90.000,B 90.000,C 0.000} C_DIS
LIN {X 108.551,Y -9.619,Z -114.645,A -90.000,B 90.000,C 0.000} C_DIS
LIN {X 108.693,Y -9.624,Z -115.612,A -90.000,B 90.000,C 0.000} C_DIS
LIN {X 108.948,Y -9.639,Z -117.705,A -90.000,B 90.000,C 0.000} C_DIS
LIN {X 109.043,Y -9.644,Z -118.444,A -90.000,B 90.000,C 0.000} C_DIS
LIN {X 109.313,Y -9.661,Z -120.978,A -90.000,B 90.000,C 0.000} C_DIS
LIN {X 109.342,Y -9.663,Z -121.237,A -90.000,B 90.000,C 0.000} C_DIS
LIN {X 109.589,Y -9.679,Z -123.945,A -90.000,B 90.000,C 0.000} C_DIS
LIN {X 109.785,Y -9.692,Z -126.530,A -90.000,B 90.000,C 0.000} C_DIS
LIN {X 109.934,Y -9.700,Z -129.128,A -90.000,B 90.000,C 0.000} C_DIS
LIN {X 109.956,Y -9.700,Z -129.550,A -90.000,B 90.000,C 0.000} C_DIS
LIN {X 110.055,Y -9.704,Z -132.202,A -90.000,B 90.000,C 0.000} C_DIS
LIN {X 110.092,Y -9.704,Z -134.108,A -90.000,B 90.000,C 0.000} C_DIS
LIN {X 110.110,Y -9.704,Z -135.059,A -90.000,B 90.000,C 0.000} C_DIS
LIN {X 110.119,Y -9.702,Z -138.220,A -90.000,B 90.000,C 0.000} C_DIS
LIN {X 110.075,Y -9.700,Z -141.662,A -90.000,B 90.000,C 0.000} C_DIS
LIN {X 109.972,Y -9.701,Z -145.222,A -90.000,B 90.000,C 0.000} C_DIS
LIN {X 109.965,Y -9.700,Z -145.387,A -90.000,B 90.000,C 0.000} C_DIS
LIN {X 109.801,Y -9.707,Z -148.935,A -90.000,B 90.000,C 0.000} C_DIS
LIN {X 109.788,Y -9.706,Z -149.150,A -90.000,B 90.000,C 0.000} C_DIS
LIN {X 109.552,Y -9.723,Z -152.759,A -90.000,B 90.000,C 0.000} C_DIS
LIN {X 109.534,Y -9.722,Z -153.000,A -90.000,B 90.000,C 0.000} C_DIS
LIN {X 109.255,Y -9.738,Z -156.416,A -90.000,B 90.000,C 0.000} C_DIS
LIN {X 109.177,Y -9.738,Z -157.309,A -90.000,B 90.000,C 0.000} C_DIS
LIN {X 108.864,Y -9.758,Z -160.665,A -90.000,B 90.000,C 0.000} C_DIS
LIN {X 108.830,Y -9.760,Z -161.017,A -90.000,B 90.000,C 0.000} C_DIS
LIN {X 108.466,Y -9.784,Z -164.659,A -90.000,B 90.000,C 0.000} C_DIS
LIN {X 108.388,Y -9.791,Z -165.392,A -90.000,B 90.000,C 0.000} C_DIS
LIN {X 108.052,Y -9.812,Z -168.647,A -90.000,B 90.000,C 0.000} C_DIS
LIN {X 107.656,Y -9.834,Z -172.329,A -90.000,B 90.000,C 0.000} C_DIS
LIN {X 107.274,Y -9.851,Z -175.678,A -90.000,B 90.000,C 0.000} C_DIS
LIN {X 106.878,Y -9.866,Z -178.912,A -90.000,B 90.000,C 0.000} C_DIS
LIN {X 106.515,Y -9.877,Z -181.645,A -90.000,B 90.000,C 0.000} C_DIS
LIN {X 106.093,Y -9.887,Z -184.603,A -90.000,B 90.000,C 0.000} C_DIS
LIN {X 105.697,Y -9.895,Z -187.221,A -90.000,B 90.000,C 0.000} C_DIS
LIN {X 105.315,Y -9.900,Z -189.654,A -90.000,B 90.000,C 0.000} C_DIS
LIN {X 104.935,Y -9.904,Z -192.027,A -90.000,B 90.000,C 0.000} C_DIS
LIN {X 104.509,Y -9.908,Z -194.595,A -90.000,B 90.000,C 0.000} C_DIS
LIN {X 103.983,Y -9.913,Z -197.629,A -90.000,B 90.000,C 0.000} C_DIS
LIN {X 103.333,Y -9.921,Z -201.241,A -90.000,B 90.000,C 0.000} C_DIS
LIN {X 102.533,Y -9.931,Z -205.538,A -90.000,B 90.000,C 0.000} C_DIS
LIN {X 101.505,Y -9.939,Z -210.747,A -90.000,B 90.000,C 0.000} C_DIS
LIN {X 100.362,Y -9.942,Z -216.113,A -90.000,B 90.000,C 0.000} C_DIS
LIN {X 99.565,Y -9.940,Z -219.522,A -90.000,B 90.000,C 0.000} C_DIS
LIN {X 99.028,Y -9.937,Z -221.832,A -90.000,B 90.000,C 0.000} C_DIS
LIN {X 98.616,Y -9.934,Z -223.434,A -90.000,B 90.000,C 0.000} C_DIS
LIN {X 98.381,Y -9.930,Z -224.337,A -90.000,B 90.000,C 0.000} C_DIS
LIN {X 97.567,Y -9.921,Z -227.441,A -90.000,B 90.000,C 0.000} C_DIS
LIN {X 97.461,Y -9.921,Z -227.829,A -90.000,B 90.000,C 0.000} C_DIS
LIN {X 96.932,Y -9.916,Z -229.696,A -90.000,B 90.000,C 0.000} C_DIS
LIN {X 96.610,Y -9.908,Z -230.814,A -90.000,B 90.000,C 0.000} C_DIS
LIN {X 95.819,Y -9.896,Z -233.531,A -90.000,B 90.000,C 0.000} C_DIS
LIN {X 95.136,Y -9.889,Z -235.736,A -90.000,B 90.000,C 0.000} C_DIS
LIN {X 94.648,Y -9.879,Z -237.290,A -90.000,B 90.000,C 0.000} C_DIS
LIN {X 93.963,Y -9.867,Z -239.437,A -90.000,B 90.000,C 0.000} C_DIS
LIN {X 92.586,Y -9.852,Z -243.561,A -90.000,B 90.000,C 0.000} C_DIS
LIN {X 92.586,Y -60.000,Z -243.561,A -90.000,B 90.000,C 0.000} C_DIS
LIN {X -120.015,Y -60.000,Z -239.602,A -90.000,B 90.000,C 0.000} C_DIS
LIN {X -120.015,Y -9.625,Z -239.602,A -90.000,B 90.000,C 0.000} C_DIS
LIN {X -119.298,Y -9.624,Z -239.115,A -90.000,B 90.000,C 0.000} C_DIS
LIN {X -117.844,Y -9.619,Z -238.137,A -90.000,B 90.000,C 0.000} C_DIS
LIN {X -110.427,Y -9.599,Z -233.200,A -90.000,B 90.000,C 0.000} C_DIS
LIN {X -102.702,Y -9.575,Z -228.141,A -90.000,B 90.000,C 0.000} C_DIS
LIN {X -94.728,Y -9.550,Z -223.010,A -90.000,B 90.000,C 0.000} C_DIS
LIN {X -91.511,Y -9.539,Z -220.985,A -90.000,B 90.000,C 0.000} C_DIS
LIN {X -86.521,Y -9.525,Z -217.844,A -90.000,B 90.000,C 0.000} C_DIS
LIN {X -83.085,Y -9.514,Z -215.733,A -90.000,B 90.000,C 0.000} C_DIS
LIN {X -80.892,Y -9.505,Z -214.393,A -90.000,B 90.000,C 0.000} C_DIS
LIN {X -78.100,Y -9.500,Z -212.691,A -90.000,B 90.000,C 0.000} C_DIS
LIN {X -76.153,Y -9.498,Z -211.513,A -90.000,B 90.000,C 0.000} C_DIS
LIN {X -70.520,Y -9.485,Z -208.136,A -90.000,B 90.000,C 0.000} C_DIS
LIN {X -69.359,Y -9.485,Z -207.439,A -90.000,B 90.000,C 0.000} C_DIS
LIN {X -67.189,Y -9.479,Z -206.144,A -90.000,B 90.000,C 0.000} C_DIS
LIN {X -63.761,Y -9.468,Z -204.108,A -90.000,B 90.000,C 0.000} C_DIS
LIN {X -61.944,Y -9.466,Z -203.031,A -90.000,B 90.000,C 0.000} C_DIS
LIN {X -59.006,Y -9.456,Z -201.263,A -90.000,B 90.000,C 0.000} C_DIS
LIN {X -57.975,Y -9.451,Z -200.649,A -90.000,B 90.000,C 0.000} C_DIS
LIN {X -55.459,Y -9.445,Z -199.149,A -90.000,B 90.000,C 0.000} C_DIS
LIN {X -54.861,Y -9.441,Z -198.797,A -90.000,B 90.000,C 0.000} C_DIS
LIN {X -54.228,Y -9.439,Z -198.409,A -90.000,B 90.000,C 0.000} C_DIS
LIN {X -52.040,Y -9.434,Z -197.057,A -90.000,B 90.000,C 0.000} C_DIS
LIN {X -49.278,Y -9.422,Z -195.348,A -90.000,B 90.000,C 0.000} C_DIS
LIN {X -46.302,Y -9.417,Z -193.422,A -90.000,B 90.000,C 0.000} C_DIS
LIN {X -44.668,Y -9.412,Z -192.364,A -90.000,B 90.000,C 0.000} C_DIS
LIN {X -44.314,Y -9.412,Z -192.125,A -90.000,B 90.000,C 0.000} C_DIS
LIN {X -42.659,Y -9.410,Z -190.999,A -90.000,B 90.000,C 0.000} C_DIS
LIN {X -40.679,Y -9.404,Z -189.650,A -90.000,B 90.000,C 0.000} C_DIS
LIN {X -40.245,Y -9.403,Z -189.343,A -90.000,B 90.000,C 0.000} C_DIS
LIN {X -39.012,Y -9.403,Z -188.465,A -90.000,B 90.000,C 0.000} C_DIS
LIN {X -37.201,Y -9.398,Z -187.173,A -90.000,B 90.000,C 0.000} C_DIS
LIN {X -36.751,Y -9.397,Z -186.841,A -90.000,B 90.000,C 0.000} C_DIS
LIN {X -34.632,Y -9.395,Z -185.279,A -90.000,B 90.000,C 0.000} C_DIS
LIN {X -34.004,Y -9.394,Z -184.820,A -90.000,B 90.000,C 0.000} C_DIS
LIN {X -33.413,Y -9.393,Z -184.363,A -90.000,B 90.000,C 0.000} C_DIS
LIN {X -31.432,Y -9.392,Z -182.837,A -90.000,B 90.000,C 0.000} C_DIS
LIN {X -31.220,Y -9.394,Z -182.666,A -90.000,B 90.000,C 0.000} C_DIS
LIN {X -28.993,Y -9.393,Z -180.844,A -90.000,B 90.000,C 0.000} C_DIS
LIN {X -28.751,Y -9.391,Z -180.647,A -90.000,B 90.000,C 0.000} C_DIS
LIN {X -26.430,Y -9.391,Z -178.599,A -90.000,B 90.000,C 0.000} C_DIS
LIN {X -24.514,Y -9.392,Z -176.745,A -90.000,B 90.000,C 0.000} C_DIS
LIN {X -24.438,Y -9.394,Z -176.661,A -90.000,B 90.000,C 0.000} C_DIS
LIN {X -22.731,Y -9.398,Z -174.806,A -90.000,B 90.000,C 0.000} C_DIS
LIN {X -22.579,Y -9.404,Z -174.618,A -90.000,B 90.000,C 0.000} C_DIS
LIN {X -22.243,Y -9.404,Z -174.200,A -90.000,B 90.000,C 0.000} C_DIS
LIN {X -21.159,Y -9.409,Z -172.854,A -90.000,B 90.000,C 0.000} C_DIS
LIN {X -21.053,Y -9.414,Z -172.700,A -90.000,B 90.000,C 0.000} C_DIS
LIN {X -20.513,Y -9.416,Z -171.921,A -90.000,B 90.000,C 0.000} C_DIS
LIN {X -19.911,Y -9.422,Z -171.055,A -90.000,B 90.000,C 0.000} C_DIS
LIN {X -19.800,Y -9.423,Z -170.896,A -90.000,B 90.000,C 0.000} C_DIS
LIN {X -19.618,Y -9.433,Z -170.593,A -90.000,B 90.000,C 0.000} C_DIS
LIN {X -19.252,Y -9.437,Z -169.979,A -90.000,B 90.000,C 0.000} C_DIS
LIN {X -18.457,Y -9.444,Z -168.640,A -90.000,B 90.000,C 0.000} C_DIS
LIN {X -18.346,Y -9.451,Z -168.425,A -90.000,B 90.000,C 0.000} C_DIS
LIN {X -18.034,Y -9.454,Z -167.811,A -90.000,B 90.000,C 0.000} C_DIS
LIN {X -17.361,Y -9.458,Z -166.503,A -90.000,B 90.000,C 0.000} C_DIS
LIN {X -17.211,Y -9.468,Z -166.159,A -90.000,B 90.000,C 0.000} C_DIS
LIN {X -16.505,Y -9.469,Z -164.490,A -90.000,B 90.000,C 0.000} C_DIS
LIN {X -16.406,Y -9.482,Z -164.185,A -90.000,B 90.000,C 0.000} C_DIS
LIN {X -16.040,Y -9.474,Z -162.980,A -90.000,B 90.000,C 0.000} C_DIS
LIN {X -16.002,Y -9.491,Z -162.730,A -90.000,B 90.000,C 0.000} C_DIS
LIN {X -15.924,Y -9.481,Z -162.085,A -90.000,B 90.000,C 0.000} C_DIS
LIN {X -15.953,Y -9.474,Z -161.773,A -90.000,B 90.000,C 0.000} C_DIS
LIN {X -15.975,Y -9.458,Z -161.594,A -90.000,B 90.000,C 0.000} C_DIS
LIN {X -16.065,Y -9.454,Z -161.307,A -90.000,B 90.000,C 0.000} C_DIS
LIN {X -16.132,Y -9.439,Z -161.111,A -90.000,B 90.000,C 0.000} C_DIS
LIN {X -16.173,Y -9.437,Z -161.026,A -90.000,B 90.000,C 0.000} C_DIS
LIN {X -16.434,Y -9.434,Z -160.472,A -90.000,B 90.000,C 0.000} C_DIS
LIN {X -16.577,Y -9.422,Z -160.175,A -90.000,B 90.000,C 0.000} C_DIS
LIN {X -16.767,Y -9.411,Z -159.807,A -90.000,B 90.000,C 0.000} C_DIS
LIN {X -16.951,Y -9.410,Z -159.450,A -90.000,B 90.000,C 0.000} C_DIS
LIN {X -17.044,Y -9.401,Z -159.274,A -90.000,B 90.000,C 0.000} C_DIS
LIN {X -17.284,Y -9.393,Z -158.895,A -90.000,B 90.000,C 0.000} C_DIS
LIN {X -17.644,Y -9.389,Z -158.321,A -90.000,B 90.000,C 0.000} C_DIS
LIN {X -17.731,Y -9.385,Z -158.185,A -90.000,B 90.000,C 0.000} C_DIS
LIN {X -18.395,Y -9.372,Z -157.316,A -90.000,B 90.000,C 0.000} C_DIS
LIN {X -18.742,Y -9.372,Z -156.860,A -90.000,B 90.000,C 0.000} C_DIS
LIN {X -18.782,Y -9.371,Z -156.808,A -90.000,B 90.000,C 0.000} C_DIS
LIN {X -18.985,Y -9.369,Z -156.587,A -90.000,B 90.000,C 0.000} C_DIS
LIN {X -19.848,Y -9.359,Z -155.616,A -90.000,B 90.000,C 0.000} C_DIS
LIN {X -20.444,Y -9.357,Z -154.943,A -90.000,B 90.000,C 0.000} C_DIS
LIN {X -20.590,Y -9.357,Z -154.803,A -90.000,B 90.000,C 0.000} C_DIS
LIN {X -22.199,Y -9.346,Z -153.178,A -90.000,B 90.000,C 0.000} C_DIS
LIN {X -22.963,Y -9.346,Z -152.406,A -90.000,B 90.000,C 0.000} C_DIS
LIN {X -23.190,Y -9.346,Z -152.182,A -90.000,B 90.000,C 0.000} C_DIS
LIN {X -25.121,Y -9.337,Z -150.218,A -90.000,B 90.000,C 0.000} C_DIS
LIN {X -26.019,Y -9.337,Z -149.303,A -90.000,B 90.000,C 0.000} C_DIS
LIN {X -26.821,Y -9.336,Z -148.439,A -90.000,B 90.000,C 0.000} C_DIS
LIN {X -29.289,Y -9.330,Z -145.723,A -90.000,B 90.000,C 0.000} C_DIS
LIN {X -29.467,Y -9.330,Z -145.519,A -90.000,B 90.000,C 0.000} C_DIS
LIN {X -29.609,Y -9.330,Z -145.352,A -90.000,B 90.000,C 0.000} C_DIS
LIN {X -30.266,Y -9.330,Z -144.534,A -90.000,B 90.000,C 0.000} C_DIS
LIN {X -32.617,Y -9.325,Z -141.543,A -90.000,B 90.000,C 0.000} C_DIS
LIN {X -32.895,Y -9.325,Z -141.144,A -90.000,B 90.000,C 0.000} C_DIS
LIN {X -34.776,Y -9.322,Z -138.114,A -90.000,B 90.000,C 0.000} C_DIS
LIN {X -35.439,Y -9.322,Z -137.064,A -90.000,B 90.000,C 0.000} C_DIS
LIN {X -35.675,Y -9.322,Z -136.637,A -90.000,B 90.000,C 0.000} C_DIS
LIN {X -37.112,Y -9.321,Z -133.863,A -90.000,B 90.000,C 0.000} C_DIS
LIN {X -37.785,Y -9.322,Z -132.573,A -90.000,B 90.000,C 0.000} C_DIS
LIN {X -39.480,Y -9.323,Z -128.838,A -90.000,B 90.000,C 0.000} C_DIS
LIN {X -39.579,Y -9.323,Z -128.608,A -90.000,B 90.000,C 0.000} C_DIS
LIN {X -40.385,Y -9.325,Z -126.703,A -90.000,B 90.000,C 0.000} C_DIS
LIN {X -40.982,Y -9.325,Z -125.273,A -90.000,B 90.000,C 0.000} C_DIS
LIN {X -41.432,Y -9.326,Z -124.219,A -90.000,B 90.000,C 0.000} C_DIS
LIN {X -41.845,Y -9.328,Z -123.270,A -90.000,B 90.000,C 0.000} C_DIS
LIN {X -42.435,Y -9.330,Z -122.036,A -90.000,B 90.000,C 0.000} C_DIS
LIN {X -42.653,Y -9.330,Z -121.588,A -90.000,B 90.000,C 0.000} C_DIS
LIN {X -43.277,Y -9.331,Z -120.516,A -90.000,B 90.000,C 0.000} C_DIS
LIN {X -43.397,Y -9.330,Z -120.312,A -90.000,B 90.000,C 0.000} C_DIS
LIN {X -44.313,Y -9.330,Z -119.007,A -90.000,B 90.000,C 0.000} C_DIS
LIN {X -45.247,Y -9.329,Z -117.817,A -90.000,B 90.000,C 0.000} C_DIS
LIN {X -45.888,Y -9.328,Z -116.997,A -90.000,B 90.000,C 0.000} C_DIS
LIN {X -47.666,Y -9.325,Z -114.811,A -90.000,B 90.000,C 0.000} C_DIS
LIN {X -47.948,Y -9.325,Z -114.472,A -90.000,B 90.000,C 0.000} C_DIS
LIN {X -49.630,Y -9.324,Z -112.413,A -90.000,B 90.000,C 0.000} C_DIS
LIN {X -50.195,Y -9.324,Z -111.733,A -90.000,B 90.000,C 0.000} C_DIS
LIN {X -50.374,Y -9.323,Z -111.509,A -90.000,B 90.000,C 0.000} C_DIS
LIN {X -51.688,Y -9.323,Z -109.863,A -90.000,B 90.000,C 0.000} C_DIS
LIN {X -52.578,Y -9.323,Z -108.759,A -90.000,B 90.000,C 0.000} C_DIS
LIN {X -53.849,Y -9.322,Z -107.085,A -90.000,B 90.000,C 0.000} C_DIS
LIN {X -54.971,Y -9.323,Z -105.612,A -90.000,B 90.000,C 0.000} C_DIS
LIN {X -56.753,Y -9.325,Z -103.221,A -90.000,B 90.000,C 0.000} C_DIS
LIN {X -57.316,Y -9.326,Z -102.473,A -90.000,B 90.000,C 0.000} C_DIS
LIN {X -58.919,Y -9.331,Z -100.366,A -90.000,B 90.000,C 0.000} C_DIS
LIN {X -59.636,Y -9.333,Z -99.420,A -90.000,B 90.000,C 0.000} C_DIS
LIN {X -59.858,Y -9.336,Z -99.146,A -90.000,B 90.000,C 0.000} C_DIS
LIN {X -61.754,Y -9.344,Z -96.816,A -90.000,B 90.000,C 0.000} C_DIS
LIN {X -62.153,Y -9.354,Z -96.381,A -90.000,B 90.000,C 0.000} C_DIS
LIN {X -63.412,Y -9.361,Z -95.018,A -90.000,B 90.000,C 0.000} C_DIS
LIN {X -63.760,Y -9.364,Z -94.637,A -90.000,B 90.000,C 0.000} C_DIS
LIN {X -64.097,Y -9.375,Z -94.314,A -90.000,B 90.000,C 0.000} C_DIS
LIN {X -65.291,Y -9.385,Z -93.178,A -90.000,B 90.000,C 0.000} C_DIS
LIN {X -65.652,Y -9.386,Z -92.828,A -90.000,B 90.000,C 0.000} C_DIS
LIN {X -66.014,Y -9.399,Z -92.519,A -90.000,B 90.000,C 0.000} C_DIS
LIN {X -67.080,Y -9.408,Z -91.621,A -90.000,B 90.000,C 0.000} C_DIS
LIN {X -67.568,Y -9.415,Z -91.209,A -90.000,B 90.000,C 0.000} C_DIS
LIN {X -67.710,Y -9.416,Z -91.085,A -90.000,B 90.000,C 0.000} C_DIS
LIN {X -67.908,Y -9.423,Z -90.932,A -90.000,B 90.000,C 0.000} C_DIS
LIN {X -69.307,Y -9.434,Z -89.870,A -90.000,B 90.000,C 0.000} C_DIS
LIN {X -69.677,Y -9.435,Z -89.581,A -90.000,B 90.000,C 0.000} C_DIS
LIN {X -69.893,Y -9.442,Z -89.426,A -90.000,B 90.000,C 0.000} C_DIS
LIN {X -70.346,Y -9.447,Z -89.108,A -90.000,B 90.000,C 0.000} C_DIS
LIN {X -71.832,Y -9.456,Z -88.067,A -90.000,B 90.000,C 0.000} C_DIS
LIN {X -72.247,Y -9.461,Z -87.790,A -90.000,B 90.000,C 0.000} C_DIS
LIN {X -73.745,Y -9.469,Z -86.800,A -90.000,B 90.000,C 0.000} C_DIS
LIN {X -73.948,Y -9.471,Z -86.668,A -90.000,B 90.000,C 0.000} C_DIS
LIN {X -75.418,Y -9.473,Z -85.730,A -90.000,B 90.000,C 0.000} C_DIS
LIN {X -75.831,Y -9.475,Z -85.469,A -90.000,B 90.000,C 0.000} C_DIS
LIN {X -77.696,Y -9.472,Z -84.294,A -90.000,B 90.000,C 0.000} C_DIS
LIN {X -78.587,Y -9.466,Z -83.719,A -90.000,B 90.000,C 0.000} C_DIS
LIN {X -79.274,Y -9.459,Z -83.272,A -90.000,B 90.000,C 0.000} C_DIS
LIN {X -79.560,Y -9.456,Z -83.082,A -90.000,B 90.000,C 0.000} C_DIS
LIN {X -80.523,Y -9.449,Z -82.433,A -90.000,B 90.000,C 0.000} C_DIS
LIN {X -81.001,Y -9.445,Z -82.105,A -90.000,B 90.000,C 0.000} C_DIS
LIN {X -81.575,Y -9.438,Z -81.692,A -90.000,B 90.000,C 0.000} C_DIS
LIN {X -82.182,Y -9.431,Z -81.247,A -90.000,B 90.000,C 0.000} C_DIS
LIN {X -82.566,Y -9.424,Z -80.947,A -90.000,B 90.000,C 0.000} C_DIS
LIN {X -83.621,Y -9.415,Z -80.111,A -90.000,B 90.000,C 0.000} C_DIS
LIN {X -84.016,Y -9.409,Z -79.776,A -90.000,B 90.000,C 0.000} C_DIS
LIN {X -84.302,Y -9.408,Z -79.531,A -90.000,B 90.000,C 0.000} C_DIS
LIN {X -84.730,Y -9.407,Z -79.163,A -90.000,B 90.000,C 0.000} C_DIS
LIN {X -85.333,Y -9.405,Z -78.634,A -90.000,B 90.000,C 0.000} C_DIS
LIN {X -85.545,Y -9.405,Z -78.448,A -90.000,B 90.000,C 0.000} C_DIS
LIN {X -86.536,Y -9.407,Z -77.594,A -90.000,B 90.000,C 0.000} C_DIS
LIN {X -86.878,Y -9.412,Z -77.319,A -90.000,B 90.000,C 0.000} C_DIS
LIN {X -87.094,Y -9.412,Z -77.148,A -90.000,B 90.000,C 0.000} C_DIS
LIN {X -87.418,Y -9.420,Z -76.922,A -90.000,B 90.000,C 0.000} C_DIS
LIN {X -87.805,Y -9.418,Z -76.656,A -90.000,B 90.000,C 0.000} C_DIS
LIN {X -88.082,Y -9.423,Z -76.486,A -90.000,B 90.000,C 0.000} C_DIS
LIN {X -88.287,Y -9.422,Z -76.364,A -90.000,B 90.000,C 0.000} C_DIS
LIN {X -88.524,Y -9.422,Z -76.225,A -90.000,B 90.000,C 0.000} C_DIS
LIN {X -88.810,Y -9.426,Z -76.073,A -90.000,B 90.000,C 0.000} C_DIS
LIN {X -89.137,Y -9.425,Z -75.902,A -90.000,B 90.000,C 0.000} C_DIS
LIN {X -89.352,Y -9.427,Z -75.801,A -90.000,B 90.000,C 0.000} C_DIS
LIN {X -89.730,Y -9.426,Z -75.625,A -90.000,B 90.000,C 0.000} C_DIS
LIN {X -90.150,Y -9.430,Z -75.448,A -90.000,B 90.000,C 0.000} C_DIS
LIN {X -90.396,Y -9.430,Z -75.345,A -90.000,B 90.000,C 0.000} C_DIS
LIN {X -90.740,Y -9.434,Z -75.221,A -90.000,B 90.000,C 0.000} C_DIS
LIN {X -90.924,Y -9.439,Z -75.168,A -90.000,B 90.000,C 0.000} C_DIS
